(* Close file and validate data *)
SysFileClose(File:=hFile);
END_ACTION
ACTION DB_SetName:
(* Create current filename 'yyyyCRnn.DAT' *)
sFile:=CONCAT(FilesPath,WORD_TO_STRING(Sys.Time_Year));
sFile:=CONCAT(STR1:=sFile, STR2:='CR');
IF ID<10 THEN
sFile:=CONCAT(STR1:=sFile, STR2:='0');
END_IF
sFile:=CONCAT(STR1:=sFile, STR2:=BYTE_TO_STRING(ID));
sFile:=CONCAT(STR1:=sFile, STR2:='.DAT');
END_ACTION
ACTION Init:
DB_Load();
InitOK:=TRUE;
END_ACTION

(* POU Plant_Objects/obj_CTL, ST *)
FUNCTION_BLOCK obj_CTL
(* === PULSE VOLUME COUNTER ===
   v1.0[16/04/15] - Versioning
*)
VAR_INPUT
	(* Settings *)
	ID				: BYTE;	(* Index of instanced object *)
	Peso			: DWORD;
	(* Physical inputs *)
	CTL_ST			: BOOL;
END_VAR
VAR_IN_OUT
	COUNT			: DWORD;
END_VAR
VAR_OUTPUT
	(* Status *)
	Status_Log		: BYTE;
END_VAR
VAR
	Filter			: FLT_TAP := ( INITEV:=FALSE );
	Timer			: TON;
	TCount			: DWORD;
	i				: DWORD;
END_VAR
(* Execute timer *)
Timer(IN:=NOT Timer.Q, PT:=T#60m);

(* Execute filter on counter status *)
Filter(IN:=CTL_ST);

(* Count event *)
IF Filter.EVH THEN
	COUNT:=COUNT+Peso;
	TCount:=TCount+1;
	(* Check flow rate *)
	IF TCount>=Plant_MaxWaterLoss THEN
		i:=(TCount*TIME_TO_DWORD(Timer.PT))/TIME_TO_DWORD(Timer.ET);	(* Estimated mc per hour *)
		i:= i * Peso;

		(* NB The weight is multiplied by 10 -> Need to divide it by 10 server side *)
		LogEv(EL_AlarmStop,EO_CTL,ID,1,DWORD_TO_STRING(i));
		Status_Log:=2;

		TCount:=0;
		Timer(IN:=FALSE);
	END_IF
END_IF
(* Check timer *)
IF Timer.Q THEN
	TCount:=0;							(* One hour is elapsed *)
	IF TCount<Plant_MaxWaterLoss THEN
		Status_Log:=0;
	END_IF
END_IF
END_FUNCTION_BLOCK
ACTION AddLogData:
Logger.s1:=INSERT('&CTL=',BYTE_TO_STRING(ID),4);
IF ID<10 THEN Logger.s1:=INSERT(Logger.s1,'0',4); END_IF

Logger.s1:=CONCAT(Logger.s1,DWORD_TO_STRING(COUNT));			Logger.s1:=CONCAT(Logger.s1,';');

Logger.s1:=CONCAT(Logger.s1,WORD_TO_STRING(Status_Log));
ADDSTRING(ADR(Logger.TData), ADR(Logger.s1), Logger.TLen);
END_ACTION

(* POU Plant_Objects/obj_MODBUS, ST *)
FUNCTION_BLOCK obj_MODBUS
(* === MODBUS PROTOCOL INTERFACE ===
   v1.1[19/06/15] - Added new VARS allocation and searching
*)
VAR CONSTANT
	VARS_Max	: BYTE := 32;
END_VAR
VAR_INPUT
	(* Settings *)
	ID			: BYTE;
	COM			: BYTE;
	BAUDRATE	: COM_BAUDRATE;
	RS485		: BOOL := FALSE;

	N_STOPBits	:BYTE:=1;

	(* Interface *)
	MB_MASTER	: MODBUS_EXTENDED_MASTER;
	MB_Start	: BOOL;
	MB_Query	: typModbusExtendedQuery;
	MB_Resp		: typModbusResponse;
	MB_Lock		: BOOL;
	MB_timeOut	: TIME := t#500ms;

	(* Variables management *)
	VARS_En		: BOOL;
	VARS		: ARRAY [0..VARS_Max] OF typ_MODBUS_VAR;
	VARS_Check	: BOOL;
	VARS_Alarm	: BOOL;

	(* Variables allocation *)
	VAR_Pointer : POINTER TO ARRAY[0..99] OF WORD;
	VAR_Cfg		: POINTER TO typ_MODBUS_VAR;
END_VAR
VAR_OUTPUT
	(* Status *)
	Status_Log	: BYTE;
	Status_Vis	: DWORD;
END_VAR
VAR
	sta         : BYTE :=0;
	i			: BYTE;
	j			: BYTE;
	Alarm		: FLT_EVENT;
	
	VarTmr		: TON := (PT:=T#1s);
	VarSta		: BYTE; (* Status *)
	VarCnt		: BYTE; (* Scan counter *)
	VarRetry	: BYTE;
	VarAlarm	: BYTE; (* Last variable with errors *)
END_VAR
IF N_STOPBits=1 THEN MB_MASTER.csCOM_STOPBITS:=STOPBITS_1;END_IF
IF N_STOPBits=2 THEN MB_MASTER.csCOM_STOPBITS:=STOPBITS_2;END_IF


(** PARITY_NO **)



MB_MASTER(ENABLE:=TRUE,	ASCII_Mode:=FALSE, bCOM_PORT:=COM, cbCOM_BAUDRATE:=BAUDRATE, cpCOM_PARITY:=PARITY_EVEN,
		cbsCOM_BYTESIZE:=BS_8, cfCOM_FLOW_CONTROL:=SEL(RS485,NO_FLOW_CONTROL,HALFDUPLEX),
		tTIME_OUT:=MB_timeOut,	StartFunction:=MB_Start, ExtQuery:=MB_Query, Response:=MB_Resp);

(* Process variable management *)
IF VARS_En THEN VARS_Process(); END_IF

(* Check status *)
Alarm(IN:=(MB_MASTER.bInterfaceError<>0));
IF Alarm.EVH THEN
	LogEv(SEL(MB_MASTER.bInterfaceError<>3,EL_Wrn,EL_Alarm),EO_MODBUS,ID,1,BYTE_TO_STRING(MB_MASTER.bInterfaceError));
END_IF
IF Alarm.EVL THEN								(* Trigger a fall edge: MODBUS back working *)
	LogEv(EL_Log,EO_MODBUS,ID,2,'MODBUS_OK');
END_IF

(* Log/visu status *)
   IF Alarm.IN   THEN Status_Log:=2; Status_Vis:=COLOR_RED;
ELSIF Vars_Alarm THEN Status_Log:=1; Status_Vis:=COLOR_YELLOW;
  				 ELSE Status_Log:=0; Status_Vis:=COLOR_GREEN;
END_IF
END_FUNCTION_BLOCK
ACTION VAR_Search:
(* Search VAR with specific pointer if not found return first free VAR
	[Last VAR is not active... used as safe area...] 
*)
j:=VARS_Max;
FOR i := 0 TO VARS_Max-1 DO
	IF VARS[i].Variable=0 AND j>i THEN j:=i; END_IF
	IF VARS[i].Variable=VAR_Pointer THEN
		VAR_Cfg:=ADR(VARS[i]);
		RETURN;
	END_IF
END_FOR
VAR_Cfg:=ADR(VARS[j]);
END_ACTION
ACTION VARS_Process:
(* Update var timers *)
VarTmr(IN:=(NOT VarTmr.Q));
IF VarTmr.Q THEN
	FOR i := 0 TO VARS_Max DO
		IF VARS[i].Refresh_Cnt>0 THEN VARS[i].Refresh_Cnt:=VARS[i].Refresh_Cnt-1; END_IF
	END_FOR
	VARS_Check:=TRUE;
END_IF


(* Process status *)
CASE VarSta OF
	0: (* === Init *)
		VarCnt:=0;
		VarSta:=1;

	1: (* === Wait check signal *)
		IF VARS_Check THEN				(* Decremented "Refresh_Cnt" *)
			VARS_Check:=FALSE;
			VarCnt:=0;
			VarSta:=2;
		END_IF

	2: (* === Check loop *)
		IF NOT (MB_Lock OR MB_Start) THEN
			WHILE VarCnt<=(VARS_Max-1) AND VarSta=2 DO
				(* Check only active vars *)
				IF VARS[VarCnt].Variable<>0 THEN			(* "Variable" is a pointer to word, so if 0 no address *)
					(* Check var auto-refresh on timer checks *)
					IF VARS[VarCnt].Refresh_Time>0 AND VARS[VarCnt].Refresh_Cnt=0 THEN
						VARS[VarCnt].Refresh_Cnt:=VARS[VarCnt].Refresh_Time;
						VarSta:=3;
					END_IF
					(* Check refresh for change or request *)
					CASE VARS[VarCnt].FunCode OF
						5,6,15,16: (* Write functions *)
							IF VARS[VarCnt].Variable_Size=1 THEN
								IF VARS[VarCnt].Variable^<>VARS[VarCnt].Variable_Mirror THEN
									VARS[VarCnt].Variable_Mirror:=VARS[VarCnt].Variable^;
									VarSta:=3;
								END_IF
							ELSE
								IF VARS[VarCnt].Variable_Mirror<>0 THEN
									VARS[VarCnt].Variable_Mirror:=0;
									VarSta:=3;
								END_IF
							END_IF
						1,2,3,4: (* Read functions *)
							IF VARS[VarCnt].Variable_Mirror<>0 THEN
								VARS[VarCnt].Variable_Mirror:=0;
								VarSta:=3;
							END_IF
					END_CASE
				END_IF
				(* Process query *)
				IF VarSta=3 THEN
					MB_Lock:=TRUE;
					MB_Query.SlaveAddress:=VARS[VarCnt].SlaveAddress;
					MB_Query.FunctionCode:=VARS[VarCnt].FunCode;
					CASE VARS[VarCnt].FunCode OF
						16#5,16#6,16#F,16#10:
							MB_Query.Read_Quantity:=0;
							MB_Query.Read_StartAddress:=0;
							MB_Query.Write_StartAddress:=VARS[VarCnt].FunAddress;
							MB_Query.Write_Quantity:=VARS[VarCnt].Variable_Size;
							IF VARS[VarCnt].Variable_Size=200 THEN
								COPY_32SWAP16(VARS[VarCnt].Variable, ADR(MB_Query.Write_Data[0]));
							ELSIF VARS[VarCnt].Variable_Size>1 THEN
								MEMCPY(VARS[VarCnt].Variable, ADR(MB_Query.Write_Data[0]), 2*VARS[VarCnt].Variable_Size);
							ELSE
								MB_Query.Write_Data[0]:=VARS[VarCnt].Variable^;
							END_IF
						16#1,16#2,16#3,16#4:
							MB_Query.Read_StartAddress:=VARS[VarCnt].FunAddress;
							IF VARS[VarCnt].Variable_Size=200 THEN MB_Query.Read_Quantity:=2; ELSE
							  MB_Query.Read_Quantity:=VARS[VarCnt].Variable_Size;
							END_IF
							MB_Query.Write_StartAddress:=0;
							MB_Query.Write_Quantity:=0;
					END_CASE
					VarRetry:=0;
					MB_Start:=TRUE;
				ELSE
					VarCnt:=VarCnt+1;
				END_IF
			END_WHILE
			(* Check loop completed -> no actions *)
			IF VarSta=2 THEN VarSta:=1; END_IF
		END_IF

	3: (* === Wait & process MB response *)
		IF NOT MB_Start THEN
			IF MB_MASTER.MB_Error=0 THEN
				CASE VARS[VarCnt].FunCode OF
					1,2,3,4:
						IF VARS[VarCnt].Variable_Size=200 THEN
							COPY_32SWAP16(ADR(MB_Resp.Data), VARS[VarCnt].Variable);
						ELSIF VARS[VarCnt].Variable_Size>1 THEN
							MEMCPY(ADR(MB_Resp.Data), VARS[VarCnt].Variable, 2*VARS[VarCnt].Variable_Size);
						ELSE
							VARS[VarCnt].Variable^:=MB_Resp.Data[0];
						END_IF
				END_CASE
				MB_Lock:=FALSE;
				(* Signal error recovery *)
				IF VARS_Alarm=TRUE AND VarCnt=VarAlarm THEN
					LogEv(EL_Wrn,EO_MODBUS,ID,5,'');
					VARS_Alarm:=FALSE;
				END_IF
				(* Next var *)
				VarCnt:=VarCnt+1;
				VarSta:=2;
			ELSE
				IF VarRetry<3 THEN
					VarRetry:=VarRetry+1;
					MB_Start:=TRUE;
				ELSE
					MB_Lock:=FALSE;
					(* Signal error *)
					IF VARS_Alarm=FALSE THEN
						LogEv(EL_Wrn,EO_MODBUS,ID,3,INT_TO_STRING(MB_MASTER.MB_Error));
						VARS_Alarm:=TRUE;
						VarAlarm:=VarCnt-1;
					END_IF
					(* Next var *)
					VarCnt:=VarCnt+1;
					VarSta:=2;
				END_IF
			END_IF
		END_IF

ELSE
	VarSta:=0;
END_CASE
END_ACTION

(* POU Plant_Objects/obj_MODBUS_THAITY_ELECTA, ST *)
FUNCTION_BLOCK obj_MODBUS_THAITY_ELECTA
VAR CONSTANT
	TimeOutModBus: TON;

END_VAR
VAR_INPUT
	ID			:	BYTE;
	Address		:	BYTE;


	SetPointManuale: INT; 			(* SetPoint forazato in manuale escludendo la curva di carico *)
	AbilitaSetPointManuale : BOOL ; (* Abilita il funzionamento col set point Manaule Escludendo la curva cliamtica *)


	(* Modbus *)
	Refresh_Now	:	BOOL;			(* Richiesta di lettura stato macchina Immediata  *)
	retryErrMax	:	BYTE := 2;

	Temperatura: INT;


	STOP_REQ: BOOL;
	RUN_REQ: BOOL;
	(* Timings *)
	OnDelay		:	TIME;
	OffDelay	:	TIME;

	OnOff		: 	BOOL;

	IndirizzoDaScrivere: WORD;
	DatoDaScrivere: INT;
	ScriviDato: BOOL;
	ScriviCoil: BOOL;


	ImpMB_2SetPoint: INT;
	ImpMB_ResetFrigo: BOOL;
	ImpMB_LocRem: BOOL;
	fWriteAttivazioneComandi:BOOL;




END_VAR
VAR_IN_OUT
	ModBus		:obj_MODBUS;
	CLIM		:typ_Clima;

END_VAR
VAR_OUTPUT
	Run			:	BOOL;

	Status_Log	:	WORD;
	Status_Vis	:	DWORD;
END_VAR
VAR
	(* da diego per gestione stato stringa > 255*)
	temp :STRING(255);
	tempRaw		: ARRAY [0..MAX_SEND_TCP_CLIENT] OF BYTE;
	tempRawLen :DINT;
	longString :STRING(250);

	(* Timer manage switch on/off delay *)
	Delay		: 	TONOF;

	AllarmePDC_MB		:ARRAY [1..11] OF	FLT_EVENT;
	AllarmePDC: BOOL;

	AllarmeRemotoFLT:	FLT_EVENT;
	AllarmeRemoto: BOOL;

	state		:	INT;
	retry		:	BYTE;
	retryErr	:	BYTE;
	ReadTmr		:	TON := (PT:=T#5s);
	fModbusAlr:BOOL;

(*	retry_write	:	BYTE;
	fWriteStatus:	BOOL;
	fWriteMode	:	BOOL;
	fWriteReset	:	BOOL; *)

	SetPointCC: DINT;
	x: INT;
	ImpMB_SetPoint: INT;
	Ctrl_Run: BOOL;


	VerificaFuctionCode: INT;
	VerificaNodoLetto: INT;
	ErroreComuModBus: BOOL;
	IndiceErrore: BYTE;

	MB_BitStato: ARRAY [0..200] OF BOOL;
	MB_RegistriLetti: ARRAY [0..450] OF INT;
	MB_Moreno: ARRAY [0..450] OF INT;

	AddressRead: BYTE;
	index: BYTE;
	indexErr: BYTE;


	indirizzoDaleggere: INT;
END_VAR
(* Aggiornamento in tempo reale dei TON e TOFF funzionamento Pompa *)

Delay.PT_OF := OffDelay;
Delay.PT_ON := OnDelay + WORD_TO_TIME(1000*ID);

(* Check climatic setup *)
IF NOT CLIM.InitOK THEN Clima_Default(); END_IF;
(* Calculate Setpoint *)

	IF Temperatura>=CLIM.Points[0].X  THEN SetPointCC:=CLIM.Points[0].Y; END_IF;
	IF Temperatura>=CLIM.Points[1].X AND Temperatura<CLIM.Points[0].X THEN SetPointCC:=CLIM.Points[0].Y; END_IF;
	IF Temperatura>=CLIM.Points[2].X AND Temperatura<CLIM.Points[1].X THEN SetPointCC:=CLIM.Points[1].Y; END_IF;
	IF Temperatura>=CLIM.Points[3].X AND Temperatura<CLIM.Points[2].X THEN SetPointCC:=CLIM.Points[2].Y; END_IF;
	IF Temperatura>=CLIM.Points[4].X AND Temperatura<CLIM.Points[3].X THEN SetPointCC:=CLIM.Points[3].Y; END_IF;
	IF Temperatura<CLIM.Points[4].X THEN SetPointCC:=CLIM.Points[4].Y; END_IF;


	IF Temperatura<CLIM.Points[4].X THEN SetPointCC:=CLIM.Points[4].Y; END_IF;


(* Scelta del set point della cladaia o vien preso dalla curva cliamtica o da un riferimento esterno *)
IF AbilitaSetPointManuale THEN
	ImpMB_SetPoint:=(SetPointManuale);
ELSE
	ImpMB_SetPoint:=DINT_TO_INT(SetPointCC);
END_IF


(* Controllo Bit di funzionamento ON e OFF  *)
Ctrl_Run := OnOff;
Delay(IN:=Ctrl_Run);



IF STOP_REQ THEN Run := 1;
	ELSIF RUN_REQ THEN Run := 0;
ELSE
	Run :=Delay.OUT;
END_IF



(* Call ModBus state machine *)
Stm();

(* Check alarm	*)
CheckAlarm();
END_FUNCTION_BLOCK
ACTION AddLogData:
Logger.s1:=INSERT('&PDC=',BYTE_TO_STRING(ID),4);
IF ID<10 THEN Logger.s1:=INSERT(Logger.s1,'0',4); END_IF



Logger.s1:=CONCAT(Logger.s1,INT_TO_STRING(MB_RegistriLetti[20]));
Logger.s1:=CONCAT(Logger.s1,';');

Logger.s1:=CONCAT(Logger.s1,SEL(WORD_TO_BOOL(MB_RegistriLetti[34]),'0','100'));
Logger.s1:=CONCAT(Logger.s1,';');

Logger.s1:=CONCAT(Logger.s1,WORD_TO_STRING(Status_Log));
ADDSTRING(ADR(Logger.TData), ADR(Logger.s1), Logger.TLen);









(*
FOR tempRawLen:=0 TO MAX_SEND_TCP_CLIENT DO
                tempRaw[tempRawLen]:=0;
END_FOR

tempRawLen:=0;


temp:=Logger.s1;
ADDSTRING(ADR(tempRaw), ADR(temp), tempRawLen);

FOR x:= 1 TO 46 DO

	temp:=CONCAT(INT_TO_STRING(MB_RegistriLetti[x]),';');
	ADDSTRING(ADR(tempRaw), ADR(temp), tempRawLen);

END_FOR

temp:=CONCAT(temp,WORD_TO_STRING(Status_Log));

ADDSTRING(ADR(tempRaw), ADR(temp), tempRawLen);
ADDSTRING(ADR(Logger.TData), ADR(tempRaw), Logger.TLen); *)
END_ACTION
ACTION CheckAlarm:
(**** GEstione Log ad Evento *****)


FOR x:=1 TO 10 DO

	AllarmePDC_MB[x](IN:=WORD_TO_BOOL(MB_RegistriLetti[x+22]) );

	IF AllarmePDC_MB[x].EVH THEN
		LogEv(EL_Alarm,EO_PDC,ID,x,CONCAT ('Allarme Attivo n. ', INT_TO_STRING(x)));
	END_IF

	IF AllarmePDC_MB[x].EVL THEN
		LogEv(EL_Log,EO_PDC,ID,x,CONCAT ('Allarme Rientrato n. ', INT_TO_STRING(x)));
	END_IF

END_FOR


AllarmePDC:=FALSE;
FOR x:=1 TO 10 DO
	IF AllarmePDC_MB[x].IN THEN
		AllarmePDC:=TRUE;
	END_IF
END_FOR


	AllarmeRemotoFLT(IN:=WORD_TO_BOOL(MB_RegistriLetti[6]) );

	IF AllarmeRemotoFLT.EVH THEN
		LogEv(EL_Alarm,EO_PDC,ID,11,'Controllo_Remoto_OK');
		AllarmeRemoto:=FALSE;
	END_IF

	IF AllarmeRemotoFLT.EVL THEN
		LogEv(EL_Alarm,EO_PDC,ID,12,'Controllo_Locale_Fault');
		AllarmeRemoto:=TRUE;
	END_IF





(* Seganalzione stato Frigorifero  *)
IF ErroreComuModBus OR AllarmePDC OR AllarmeRemoto THEN
		Status_Log:=2;
		Status_Vis:=16#2020F0;
    ELSE
		Status_Log:=0;
		Status_Vis:=16#006000;
END_IF
END_ACTION
ACTION Clima_Default:
IF CLIM.Points[0].X=0 THEN
	CLIM.Points[0].X:=-300; CLIM.Points[0].Y:=770;
	CLIM.Points[1].X:=-70 ; CLIM.Points[1].Y:=770;
	CLIM.Points[2].X:= 80; 	CLIM.Points[2].Y:=690;
	CLIM.Points[3].X:= 200; CLIM.Points[3].Y:=300;
	CLIM.Points[4].X:= 500; CLIM.Points[4].Y:=200;
END_IF
CLIM.InitOK:=TRUE;
LogEv(EL_Wrn,EO_PDC,ID,0,'Climatic_default');
END_ACTION
ACTION Stm:
CASE state OF
	0:	(* Refresh time manager *)
		ReadTmr(IN:=NOT ReadTmr.Q);
		(*A tempo interrogo il nodo sempre che non ci sia qualcuno che lo sta interrogando in quel momento *)

		IF (ReadTmr.Q AND NodoDaInterrogarePDC=Address )OR Refresh_Now AND NOT InibiscoModbusPDC THEN
			state := 10;
			ReadTmr.PT := T#5s;  (* moreno *)
			Refresh_Now := FALSE;
			InibiscoModbusPDC := TRUE;
		END_IF

	(**** Leggo le Analogiche a Disposzione  ****)

	10:	(* richiedo lettura Holding Registere Chiller  *)

		Modbus.MB_Query.SlaveAddress := Address;
		Modbus.MB_Query.FunctionCode := 3;
		ModBus.MB_Query.Read_StartAddress := 8975 ;			(* richiedo lettura altri Parametri *)
		ModBus.MB_Query.Read_Quantity := 10;
		ModBus.MB_Start := TRUE;
		state := 20;

	20:	(* Risposta all'interrogazione *)
		IF NOT ModBus.MB_Start   THEN
			VerificaFuctionCode:=ModBus.MB_Resp.FunctionCode;
			VerificaNodoLetto:=ModBus.MB_Resp.SlaveAddress;

			IF ModBus.MB_MASTER.MB_Error<>0 THEN
				state := 300;
			ELSE
				MB_RegistriLetti[1] := ModBus.MB_Resp.Data[0];   	(* Vedi tabella *)
				MB_RegistriLetti[2] := ModBus.MB_Resp.Data[1];		(* Vedi tabella *)

				ModBus.MB_Query.Read_StartAddress := 8961; 	(* richiedo lettura altri Parametri *)
				ModBus.MB_Query.Read_Quantity := 18;
				ModBus.MB_Start := TRUE;

				state := 30;
			END_IF
		END_IF

	30: (* Rispota Altri paramenti *)
		IF NOT ModBus.MB_Start  THEN

			IF ModBus.MB_MASTER.MB_Error<>0 THEN
				state := 300;
			ELSE
				MB_RegistriLetti[3] := ModBus.MB_Resp.Data[0];   	(* Vedi tabella *)
				MB_RegistriLetti[4] := ModBus.MB_Resp.Data[1];		(* Vedi tabella *)
				MB_RegistriLetti[5] := ModBus.MB_Resp.Data[3];		(* Vedi tabella *)
				MB_RegistriLetti[6] := ModBus.MB_Resp.Data[4];		(* Vedi tabella *)
				MB_RegistriLetti[7] := ModBus.MB_Resp.Data[5];		(* Vedi tabella *)
				MB_RegistriLetti[8] := ModBus.MB_Resp.Data[7];		(* Vedi tabella *)
				MB_RegistriLetti[9] := ModBus.MB_Resp.Data[9];		(* Vedi tabella *)
				MB_RegistriLetti[10] := ModBus.MB_Resp.Data[10];		(* Vedi tabella *)
				MB_RegistriLetti[11] := ModBus.MB_Resp.Data[11];		(* Vedi tabella *)
				MB_RegistriLetti[12] := ModBus.MB_Resp.Data[12];		(* Vedi tabella *)
				MB_RegistriLetti[13] := ModBus.MB_Resp.Data[16];		(* Vedi tabella *)

				ModBus.MB_Query.Read_StartAddress := 8983; (* richiedo lettura altri Parametri *)
				ModBus.MB_Query.Read_Quantity := 20;
				ModBus.MB_Start := TRUE;

				state := 40;
			END_IF
		END_IF

	40: (* Rispota Altri paramenti *)
		IF NOT ModBus.MB_Start  THEN

			IF ModBus.MB_MASTER.MB_Error<>0 THEN
				state := 300;
			ELSE
				MB_RegistriLetti[14] := ModBus.MB_Resp.Data[0];   	(* Vedi tabella *)
				MB_RegistriLetti[15] := ModBus.MB_Resp.Data[2];		(* Vedi tabella *)
				MB_RegistriLetti[16] := ModBus.MB_Resp.Data[6];		(* Vedi tabella *)
				MB_RegistriLetti[17] := ModBus.MB_Resp.Data[7];		(* Vedi tabella *)
				MB_RegistriLetti[18] := ModBus.MB_Resp.Data[8];		(* Vedi tabella *)
				MB_RegistriLetti[19] := ModBus.MB_Resp.Data[9];		(* Vedi tabella *)
				MB_RegistriLetti[20] := ModBus.MB_Resp.Data[10];		(* Vedi tabella *)
				MB_RegistriLetti[21] := ModBus.MB_Resp.Data[13];		(* Vedi tabella *)
				MB_RegistriLetti[22] := ModBus.MB_Resp.Data[17];		(* Vedi tabella *)

				ModBus.MB_Query.Read_StartAddress := 9003; (* richiedo lettura altri Parametri *)
				ModBus.MB_Query.Read_Quantity := 12;
				ModBus.MB_Start := TRUE;

				state := 45;
			END_IF
		END_IF

	45: (* Rispota Altri paramenti *)
		IF NOT ModBus.MB_Start  THEN

			IF ModBus.MB_MASTER.MB_Error<>0 THEN
				state := 300;
			ELSE
				MB_RegistriLetti[23] := ModBus.MB_Resp.Data[0];   	(* Vedi tabella *)
				MB_RegistriLetti[24] := ModBus.MB_Resp.Data[1];		(* Vedi tabella *)
				MB_RegistriLetti[25] := ModBus.MB_Resp.Data[2];		(* Vedi tabella *)
				MB_RegistriLetti[26] := ModBus.MB_Resp.Data[3];		(* Vedi tabella *)
				MB_RegistriLetti[27] := ModBus.MB_Resp.Data[4];		(* Vedi tabella *)
				MB_RegistriLetti[28] := ModBus.MB_Resp.Data[5];		(* Vedi tabella *)
				MB_RegistriLetti[29] := ModBus.MB_Resp.Data[6];		(* Vedi tabella *)
				MB_RegistriLetti[30] := ModBus.MB_Resp.Data[7];		(* Vedi tabella *)
				MB_RegistriLetti[31] := ModBus.MB_Resp.Data[9];		(* Vedi tabella *)
				MB_RegistriLetti[32] := ModBus.MB_Resp.Data[10];		(* Vedi tabella *)

				ModBus.MB_Query.Read_StartAddress := 16383; (* richiedo lettura altri Parametri *)
				ModBus.MB_Query.Read_Quantity := 20;
				ModBus.MB_Start := TRUE;

				state := 50;
			END_IF
		END_IF
	50: (* Rispota Altri paramenti *)
		IF NOT ModBus.MB_Start  THEN

			IF ModBus.MB_MASTER.MB_Error<>0 THEN
				state := 300;
			ELSE
				MB_RegistriLetti[33] := ModBus.MB_Resp.Data[0];   	(* Vedi tabella *)
				MB_RegistriLetti[34] := ModBus.MB_Resp.Data[1];		(* Vedi tabella *)
				MB_RegistriLetti[35] := ModBus.MB_Resp.Data[2];		(* Vedi tabella *)
				MB_RegistriLetti[36] := ModBus.MB_Resp.Data[3];		(* Vedi tabella *)
				MB_RegistriLetti[37] := ModBus.MB_Resp.Data[4];		(* Vedi tabella *)
				MB_RegistriLetti[38] := ModBus.MB_Resp.Data[5];		(* Vedi tabella *)
				MB_RegistriLetti[39] := ModBus.MB_Resp.Data[6];		(* Vedi tabella *)
				MB_RegistriLetti[40] := ModBus.MB_Resp.Data[8];		(* Vedi tabella *)
				MB_RegistriLetti[41] := ModBus.MB_Resp.Data[9];		(* Vedi tabella *)
				MB_RegistriLetti[42] := ModBus.MB_Resp.Data[11];		(* Vedi tabella *)
				MB_RegistriLetti[43] := ModBus.MB_Resp.Data[12];		(* Vedi tabella *)
				MB_RegistriLetti[44] := ModBus.MB_Resp.Data[13];		(* Vedi tabella *)
				MB_RegistriLetti[45] := ModBus.MB_Resp.Data[14];		(* Vedi tabella *)
				MB_RegistriLetti[46] := ModBus.MB_Resp.Data[15];		(* Vedi tabella *)

				ModBus.MB_Query.Read_StartAddress := 16399; (* richiedo lettura altri Parametri *)
				ModBus.MB_Query.Read_Quantity := 20;
				ModBus.MB_Start := TRUE;

				state := 55;
			END_IF
		END_IF

	55: (* Rispota Altri paramenti *)
		IF NOT ModBus.MB_Start  THEN

			IF ModBus.MB_MASTER.MB_Error<>0 THEN
				state := 300;
			ELSE
				MB_RegistriLetti[47] := ModBus.MB_Resp.Data[0];   	(* Vedi tabella *)
				MB_RegistriLetti[48] := ModBus.MB_Resp.Data[1];		(* Vedi tabella *)
				MB_RegistriLetti[49] := ModBus.MB_Resp.Data[2];		(* Vedi tabella *)
				MB_RegistriLetti[50] := ModBus.MB_Resp.Data[3];		(* Vedi tabella *)
				MB_RegistriLetti[51] := ModBus.MB_Resp.Data[4];		(* Vedi tabella *)
				MB_RegistriLetti[52] := ModBus.MB_Resp.Data[5];		(* Vedi tabella *)
				MB_RegistriLetti[53] := ModBus.MB_Resp.Data[6];		(* Vedi tabella *)
				MB_RegistriLetti[54] := ModBus.MB_Resp.Data[7];		(* Vedi tabella *)
				MB_RegistriLetti[55] := ModBus.MB_Resp.Data[8];		(* Vedi tabella *)
				MB_RegistriLetti[56] := ModBus.MB_Resp.Data[9];		(* Vedi tabella *)
				MB_RegistriLetti[57] := ModBus.MB_Resp.Data[10];		(* Vedi tabella *)
				MB_RegistriLetti[58] := ModBus.MB_Resp.Data[11];		(* Vedi tabella *)
				MB_RegistriLetti[59] := ModBus.MB_Resp.Data[12];		(* Vedi tabella *)
				MB_RegistriLetti[60] := ModBus.MB_Resp.Data[13];		(* Vedi tabella *)
				MB_RegistriLetti[61] := ModBus.MB_Resp.Data[14];		(* Vedi tabella *)
				MB_RegistriLetti[62] := ModBus.MB_Resp.Data[15];		(* Vedi tabella *)
				MB_RegistriLetti[63] := ModBus.MB_Resp.Data[16];		(* Vedi tabella *)
				MB_RegistriLetti[64] := ModBus.MB_Resp.Data[17];		(* Vedi tabella *)
				MB_RegistriLetti[65] := ModBus.MB_Resp.Data[18];		(* Vedi tabella *)
				MB_RegistriLetti[66] := ModBus.MB_Resp.Data[19];		(* Vedi tabella *)

				ModBus.MB_Query.Read_StartAddress := 16419; (* richiedo lettura altri Parametri *)
				ModBus.MB_Query.Read_Quantity := 20;
				ModBus.MB_Start := TRUE;

				state := 60;
			END_IF
		END_IF

	60: (* Rispota Altri paramenti *)
		IF NOT ModBus.MB_Start  THEN

			IF ModBus.MB_MASTER.MB_Error<>0 THEN
				state := 300;
			ELSE
				MB_RegistriLetti[67] := ModBus.MB_Resp.Data[0];   	(* Vedi tabella *)
				MB_RegistriLetti[68] := ModBus.MB_Resp.Data[1];		(* Vedi tabella *)
				MB_RegistriLetti[69] := ModBus.MB_Resp.Data[2];		(* Vedi tabella *)
				MB_RegistriLetti[70] := ModBus.MB_Resp.Data[3];		(* Vedi tabella *)
				MB_RegistriLetti[71] := ModBus.MB_Resp.Data[4];		(* Vedi tabella *)
				MB_RegistriLetti[72] := ModBus.MB_Resp.Data[5];		(* Vedi tabella *)
				MB_RegistriLetti[73] := ModBus.MB_Resp.Data[6];		(* Vedi tabella *)
				MB_RegistriLetti[74] := ModBus.MB_Resp.Data[7];		(* Vedi tabella *)
				MB_RegistriLetti[75] := ModBus.MB_Resp.Data[8];		(* Vedi tabella *)
				MB_RegistriLetti[76] := ModBus.MB_Resp.Data[9];		(* Vedi tabella *)
				MB_RegistriLetti[77] := ModBus.MB_Resp.Data[10];		(* Vedi tabella *)
				MB_RegistriLetti[78] := ModBus.MB_Resp.Data[11];		(* Vedi tabella *)
				MB_RegistriLetti[79] := ModBus.MB_Resp.Data[12];		(* Vedi tabella *)
				MB_RegistriLetti[80] := ModBus.MB_Resp.Data[13];		(* Vedi tabella *)
				MB_RegistriLetti[81] := ModBus.MB_Resp.Data[14];		(* Vedi tabella *)
				MB_RegistriLetti[82] := ModBus.MB_Resp.Data[15];		(* Vedi tabella *)
				MB_RegistriLetti[83] := ModBus.MB_Resp.Data[16];		(* Vedi tabella *)

				ModBus.MB_Query.Read_StartAddress := 16442; (* richiedo lettura altri Parametri *)
				ModBus.MB_Query.Read_Quantity := 10;
				ModBus.MB_Start := TRUE;

				state := 65;
			END_IF
		END_IF

	65: (* Rispota Altri paramenti *)
		IF NOT ModBus.MB_Start  THEN

			IF ModBus.MB_MASTER.MB_Error<>0 THEN
				state := 300;
			ELSE
				MB_RegistriLetti[84] := ModBus.MB_Resp.Data[0];   	(* Vedi tabella *)
				MB_RegistriLetti[85] := ModBus.MB_Resp.Data[1];		(* Vedi tabella *)
				MB_RegistriLetti[86] := ModBus.MB_Resp.Data[2];		(* Vedi tabella *)
				MB_RegistriLetti[87] := ModBus.MB_Resp.Data[3];		(* Vedi tabella *)
				MB_RegistriLetti[88] := ModBus.MB_Resp.Data[4];		(* Vedi tabella *)

				ModBus.MB_Query.Read_StartAddress := 16451; (* richiedo lettura altri Parametri *)
				ModBus.MB_Query.Read_Quantity := 20;
				ModBus.MB_Start := TRUE;

				state := 70;
			END_IF
		END_IF

	70: (* Rispota Altri paramenti *)
		IF NOT ModBus.MB_Start  THEN

			IF ModBus.MB_MASTER.MB_Error<>0 THEN
				state := 300;
			ELSE
				MB_RegistriLetti[89] := ModBus.MB_Resp.Data[0];   	(* Vedi tabella *)
				MB_RegistriLetti[90] := ModBus.MB_Resp.Data[1];		(* Vedi tabella *)
				MB_RegistriLetti[91] := ModBus.MB_Resp.Data[2];		(* Vedi tabella *)
				MB_RegistriLetti[92] := ModBus.MB_Resp.Data[3];		(* Vedi tabella *)
				MB_RegistriLetti[93] := ModBus.MB_Resp.Data[4];		(* Vedi tabella *)
				MB_RegistriLetti[94] := ModBus.MB_Resp.Data[5];		(* Vedi tabella *)
				MB_RegistriLetti[95] := ModBus.MB_Resp.Data[6];		(* Vedi tabella *)
				MB_RegistriLetti[96] := ModBus.MB_Resp.Data[7];		(* Vedi tabella *)
				MB_RegistriLetti[97] := ModBus.MB_Resp.Data[8];		(* Vedi tabella *)
				MB_RegistriLetti[98] := ModBus.MB_Resp.Data[9];		(* Vedi tabella *)
				MB_RegistriLetti[99] := ModBus.MB_Resp.Data[10];		(* Vedi tabella *)
				MB_RegistriLetti[100] := ModBus.MB_Resp.Data[11];		(* Vedi tabella *)
				MB_RegistriLetti[101] := ModBus.MB_Resp.Data[12];		(* Vedi tabella *)
				MB_RegistriLetti[102] := ModBus.MB_Resp.Data[13];		(* Vedi tabella *)
				MB_RegistriLetti[103] := ModBus.MB_Resp.Data[14];		(* Vedi tabella *)
				MB_RegistriLetti[104] := ModBus.MB_Resp.Data[15];		(* Vedi tabella *)
				MB_RegistriLetti[105] := ModBus.MB_Resp.Data[16];		(* Vedi tabella *)

				ModBus.MB_Query.Read_StartAddress := 16487; (* richiedo lettura altri Parametri *)
				ModBus.MB_Query.Read_Quantity := 2;
				ModBus.MB_Start := TRUE;

				state := 75;
			END_IF
		END_IF


	75: (* Rispota Altri paramenti *)
		IF NOT ModBus.MB_Start  THEN

			IF ModBus.MB_MASTER.MB_Error<>0 THEN
				state := 300;
			ELSE
				MB_RegistriLetti[106] := ModBus.MB_Resp.Data[0];   	(* Vedi tabella *)

				state := 200;
			END_IF
		END_IF



	100: (* Rispota Altri paramenti *)
		IF NOT ModBus.MB_Start  THEN

			IF ModBus.MB_MASTER.MB_Error<>0 THEN
				state := 300;
			ELSE
				ModBus.MB_Query.Read_StartAddress := indirizzoDaleggere; (* richiedo lettura altri Parametri *)
				ModBus.MB_Query.Read_Quantity := 4;
				ModBus.MB_Start := TRUE;

				state := 105;
			END_IF
		END_IF


	105: (* Rispota Altri paramenti *)
		IF NOT ModBus.MB_Start  THEN

			IF ModBus.MB_MASTER.MB_Error<>0 THEN
				state := 300;
			ELSE
				MB_Moreno[1] := ModBus.MB_Resp.Data[0];   	(* Vedi tabella *)
				MB_Moreno[2] := ModBus.MB_Resp.Data[1];		(* Vedi tabella *)
				MB_Moreno[3] := ModBus.MB_Resp.Data[2];		(* Vedi tabella *)
				MB_Moreno[4] := ModBus.MB_Resp.Data[3];		(* Vedi tabella *)

				state := 200;
			END_IF
		END_IF



	200:    (* Scrittura Abilitazione  *)
		IF NOT ModBus.MB_Start THEN
			IF ModBus.MB_MASTER.MB_Error<>0 THEN (*OR ModBus.MB_MASTER.MB_Error<>0 THEN*)
				state := 300;
			ELSE
					Modbus.MB_Query.FunctionCode := 6;
					Modbus.MB_Query.SlaveAddress := Address;
					ModBus.MB_Query.Write_StartAddress := 16384;
					ModBus.MB_Query.Write_Quantity :=1;
					ModBus.MB_Query.Write_Data[0] := BOOL_TO_WORD(Run);
					ModBus.MB_Start := TRUE;
					state := 210;
				END_IF
		END_IF

	210:    (* Scrittura Set Point  *)
		IF NOT ModBus.MB_Start THEN
			IF ModBus.MB_MASTER.MB_Error<>0 THEN (*OR ModBus.MB_MASTER.MB_Error<>0 THEN*)
				state := 300;
			ELSE
				IF Run <> INT_TO_BOOL (MB_RegistriLetti[34]) THEN
					Modbus.MB_Query.FunctionCode := 6;
					Modbus.MB_Query.SlaveAddress := Address;
					ModBus.MB_Query.Write_StartAddress := 16423;
					ModBus.MB_Query.Write_Quantity :=1;
					ModBus.MB_Query.Write_Data[0] := ImpMB_SetPoint+50;
					ModBus.MB_Start := TRUE;
					state := 215;
				ELSE
					state := 215;
				END_IF
			END_IF
		END_IF
	215:    (* Scrittura Set Point  *)
		IF NOT ModBus.MB_Start THEN
			IF ModBus.MB_MASTER.MB_Error<>0 THEN (*OR ModBus.MB_MASTER.MB_Error<>0 THEN*)
				state := 300;
			ELSE
				IF Run THEN
					Modbus.MB_Query.FunctionCode := 6;
					Modbus.MB_Query.SlaveAddress := Address;
					ModBus.MB_Query.Write_StartAddress := 16424;
					ModBus.MB_Query.Write_Quantity :=1;
					ModBus.MB_Query.Write_Data[0] := ImpMB_SetPoint+50;
					ModBus.MB_Start := TRUE;
					state := 290;
				ELSE
					state := 290;
				END_IF
			END_IF
		END_IF


		290:    (* Scrittura BOOL - COIL o WORD *)
		IF NOT ModBus.MB_Start THEN
			IF ModBus.MB_MASTER.MB_Error<>0 THEN (*OR ModBus.MB_MASTER.MB_Error<>0 THEN*)
				state := 300;
			ELSE
				IF ScriviDato THEN
				(*	IF ScriviCoil THEN
						Modbus.MB_Query.FunctionCode := 5;
					ELSE
						Modbus.MB_Query.FunctionCode := 6;
					END_IF *)
					Modbus.MB_Query.FunctionCode := 6;
					Modbus.MB_Query.SlaveAddress := Address;
					ModBus.MB_Query.Write_StartAddress := IndirizzoDaScrivere - 1;
					ModBus.MB_Query.Write_Quantity :=1;
					ModBus.MB_Query.Write_Data[0] := DatoDaScrivere;
					ModBus.MB_Start := TRUE;

				MB_Moreno[10] :=  MB_Moreno[10]+1;   	(* Vedi tabella *)

				(*		IF ScriviCoil THEN
							IF 	MB_BitStato[IndirizzoDaScrivere]=WORD_TO_BOOL(DatoDaScrivere) THEN
								ScriviDato:=FALSE;
							END_IF
						ELSE
							IF 	MB_RegistriLetti[IndirizzoDaScrivere]=DatoDaScrivere THEN
								ScriviDato:=FALSE;
							END_IF
						END_IF *)
					state := 295;
				ELSE
					state := 295;
				END_IF
			END_IF
		END_IF




		295:
		IF NOT ModBus.MB_Start THEN
			IF ModBus.MB_MASTER.MB_Error<>0 THEN (*OR ModBus.MB_MASTER.MB_Error<>0 THEN*)
				state := 300;
			ELSE
				IF fModbusAlr THEN fModbusAlr := FALSE; END_IF
				NodoDaInterrogarePDC:=Address+1;
				InibiscoModbusPDC:=FALSE;
				retryErr := 0;
				retry := 0;
				state := 0;
					IF fModbusAlr=FALSE AND ErroreComuModBus=TRUE THEN
						LogEv(EL_Log,EO_PDC,ID,62,'ComunicazioneModBus_OK');
						ErroreComuModBus := FALSE;
				(*	WarningCtr := SEL(WarningCtr=0, WarningCtr-1, 0); *)
					END_IF


			END_IF
		END_IF



	(**** CHECK MODBUS ERROR ****)
	300: 	(* Release MODBUS *)
			InibiscoModbusPDC:=FALSE;
			(* Retries *)
			retry:=retry+1;
			IF retry>3 THEN
				retry:=0;

				(* Verify if slave is dead *)
				IF retryErr < retryErrMaX THEN
					retryErr := retryErr + 1;
				ELSE
					fModbusAlr := TRUE;
					(* Verify ModBus error	*)

					IF fModbusAlr AND ErroreComuModBus=FALSE THEN
						LogEv(EL_Alarm,EO_PDC,ID,61,CONCAT('ErroreModbus_',INT_TO_STRING(ModBus.MB_MASTER.MB_Error)));
						ErroreComuModBus := TRUE;
					END_IF
				END_IF

				END_IF
			Refresh_Now := FALSE;
			NodoDaInterrogarePDC:=Address+1;
			state:=0;
END_CASE




(* Controllo Time Out Ciclo ModBus *)

TimeOutModBus(In:=state<>0,PT:=t#30s);
IF TimeOutModBus.Q THEN
	State:=0;
	Refresh_Now:=TRUE;  (* Rilancio la lettura del nodo *)
	IF MODBUS.MB_Lock=TRUE THEN MODBUS.MB_Lock:=FALSE;END_IF
	IF InibiscoModbusPDC=TRUE THEN InibiscoModbusPDC:=FALSE;END_IF
END_IF
END_ACTION

(* POU Plant_Objects/obj_TPV, ST *)
FUNCTION_BLOCK obj_TPV
(* === TEMPERATURE PROBE  ===
   v1.0[16/04/15] - Versioning
*)
VAR CONSTANT
	NormalEv		: BYTE := 0;
	ErrorEv			: BYTE := 1;
	WarningEv		: BYTE := 2;
END_VAR
VAR_INPUT
	(* Settings *)
	ID				: BYTE;
	TAP				: BYTE:=4;	   (* Consecutive checks filter *)
	INITEV			: BOOL:= TRUE; (* Generate init OK event *)
	IN_EMIN			: INT :=-2000; (* Low error limit *)
	IN_WMIN			: INT := -550; (* Low warning value *)
	IN_WMAX			: INT :=  900; (* High warning value *)
	IN_EMAX			: INT := 8500; (* High error limit *)
	ERR_MIN_SHORT	: BOOL:= TRUE; (* TRUE  ==> EMIN=Short        , EMAX=Disconnected
									  FALSE ==> EMIN=Disconnected , EMAX=Short 		 *)
	(* Physical input *)
	IN			: INT;
END_VAR
VAR_OUTPUT
	WRN			: BOOL;	(* Value in warning range *)
	ERR			: BOOL;	(* Value error *)
	HI			: INT;	(* Highest value - cleared by Stat_Reset() action *)
	AVG			: INT; 	(* Average value - updated by Mean() action, cleared by Mean_Reset() action *)
	LOW			: INT;	(* Lowest value  - cleared by Stat_Reset() action *)

	Status_Log	: WORD;
	Status_Vis	: DWORD;
END_VAR
VAR
	cnt			: BYTE;
	event		: BYTE := 0;	(* 0: monitoring a generic, 1: monitoring an error, 2: monitoring a warning *)
	asum		: DINT;
	acnt		: WORD;
END_VAR
(* Check probe value limits *)
IF IN<=IN_EMIN OR IN>=IN_EMAX THEN
	IF NOT ERR THEN
		IF event <> ErrorEv THEN
			cnt := 1;
			event := ErrorEv;
		ELSE
			cnt:=cnt+1;
		END_IF

		IF cnt>TAP THEN
			cnt:=0;
			ERR:=TRUE; WRN:=FALSE;
			IF ( ERR_MIN_SHORT=TRUE  AND IN<=IN_EMIN ) OR ( ERR_MIN_SHORT=FALSE AND IN>=IN_EMAX ) THEN
				LogEv(EL_Alarm,EO_TPV,ID,5,INT_TO_STRING(IN));
			ELSE
				LogEv(EL_Alarm,EO_TPV,ID,4,INT_TO_STRING(IN));
			END_IF
		END_IF
	END_IF
ELSIF IN<=IN_WMIN OR IN>=IN_WMAX THEN
	IF NOT WRN THEN
		IF event <> WarningEv THEN
			cnt := 1;
			event := WarningEv;
		ELSE
			cnt:=cnt+1;
		END_IF

		IF cnt>TAP THEN
			cnt:=0;
			ERR:=FALSE; WRN:=TRUE;
			LogEv(EL_Wrn,EO_TPV,ID,SEL(IN<=IN_WMIN,3,2),INT_TO_STRING(IN));
		END_IF
	END_IF
ELSE
	IF INITEV OR WRN OR ERR THEN
		IF event <> NormalEv THEN
			cnt := 1;
			event := NormalEv;
		ELSE
			cnt:=cnt+1;
		END_IF

		IF cnt>TAP THEN
			cnt:=0;
			INITEV:=FALSE; ERR:=FALSE; WRN:=FALSE;
			LogEv(EL_Log,EO_TPV,ID,1,'Probe_OK');
		END_IF
	END_IF
END_IF


(*
(* Average value *)
IF acnt>=500 THEN
	Mean();
	asum := asum - AVG;
	acnt := acnt - 1;
END_IF

asum := asum + IN;
acnt := acnt + 1;
*)

AVG := IN;



(* Statistics values *)
IF IN<LOW THEN LOW:=IN; END_IF
IF IN>HI  THEN HI :=IN; END_IF



(* Status Log *)
IF ERR THEN	Status_Log := 2; Status_Vis := COLOR_RED;
ELSIF WRN THEN Status_Log := 1;	Status_Vis := COLOR_YELLOW;
ELSE Status_Log := 0; Status_Vis := COLOR_GREEN;
END_IF
END_FUNCTION_BLOCK
ACTION AddLogData:
Logger.s1:=INSERT('&TPV=',BYTE_TO_STRING(ID),4);
IF ID<10 THEN Logger.s1:=INSERT(Logger.s1,'0',4); END_IF
(*
Mean();
*)
Logger.s1:=CONCAT(Logger.s1,INT_TO_STRING(AVG));		Logger.s1:=CONCAT(Logger.s1,';');

Logger.s1:=CONCAT(Logger.s1,WORD_TO_STRING(Status_Log));
ADDSTRING(ADR(Logger.TData), ADR(Logger.s1), Logger.TLen);
END_ACTION
ACTION Mean:
AVG := DINT_TO_INT(asum/acnt);
END_ACTION
ACTION Mean_Reset:
AVG:=IN;
asum:=IN;
acnt:=1;
END_ACTION
ACTION Stat_Reset:
HI:=IN;
LOW:=IN;
END_ACTION

(* POU Plant_Objects/obj_VRD_02, ST *)
FUNCTION_BLOCK obj_VRD_02
(* === VALVOLA RIPARTITORE ===
  VERSIONE 01 REALIZZATA DA MORENO E TESTATA SU IMPIANTO SAN FELICE ID 012 CLV

			02   - 	Introdotto possibilità di impstare il set point in Automatico ( da curva Cliamtica ) o da remoto ( set Point
				 	impostato fuori dalla FB per dare un Set Point Fisso.
				 -	Introdotto Temperatura di Controllo Curva climatica con paramentro di ingresso delle FB 



*)
VAR CONSTANT
	Chk_CntSecAlarm	: INT := 900;	(* 900s = 15 minutes -> Observation itme *)
END_VAR

VAR_INPUT
	(* Settings *)
	ID				: BYTE;
	(* Controls *)
	RUN  			: BOOL;					(* Control input *)
	ReducedRange	: BOOL := FALSE;		(* If true output value is among 2 and 10V, otherwise 0-10V *)

	(* Physical inputs *)
	TEMP 			: INT;		(* Input temperature from sensor *)
	STATUS 			: WORD;		(* Input position from valve *)

	InitOK			: BOOL;
	Alarm1			: BOOL;
	Alarm2			: BOOL;
	Warning			: BOOL;

	Ctrl_Init		: BOOL;
	Ctrl_SetPoint	: INT;
	Ctrl_SetPointNew: INT := 0;
	Delta_SetPoint	: INT;
	Ctrl_Err		: INT;			(* Current error *)
	Ctrl_Err0		: INT; 			(* Previous error *)
	Ctrl_Accel		: REAL;			(* Derivate of error *)
	Ctrl_AccelGate  : INT:=1;		(* Derivate gate *)
	Ctrl_AccelTmr	: WORD;
	Ctrl_SetPointGate: INT := 5;	(* Setpoint gate - 0.5°C *)
	Ctrl_Out		: REAL;

	Chk_Err			: INT;
	Chk_Cnt			: INT;
	Chk_CntAlarm	: INT:=240; 		(* Check error trigger 120s *)

	(* Status *)
	Log_AvgTemp		: AVERAGE_T;
	Status_Log		: BYTE;
	Status_Vis 		: DWORD;

	(* Feedback *)
	fFeedback		: BOOL;			(* TRUE: Feedback available, FALSE: Feedback not available *)

	OffsetBoost: INT;

	ComandoManuale:BOOL:=FALSE;
	RiferimentoManuale:INT;

	TempControlloCC:INT;

	AbilitaSetPointManuale: BOOL:=FALSE;
	SetPointManuale: INT:=400;


END_VAR
VAR_IN_OUT
	CLIM		: typ_Clima;
END_VAR
VAR_OUTPUT
	(* Physical outputs *)
	OUT			: WORD;
END_VAR
VAR
	Curve		: CHARCURVE;
	Curve_Err	: BYTE;

	aTemp		: ARRAY [1..20] OF INT;
	meanTemp	: INT;
	sum			: INT := 0;
	Tmr			: TON := (PT:=T#1s);
	index		: BYTE;
	i			: BYTE;
	fCtrl_Err	: BOOL;		(* TRUE: Ctrl_Err>0, FALSE: Ctrl_Err<0 *)

	SetPoint: INT;
END_VAR

VAR_INPUT RETAIN
	Ctrl_ErrGate	: INT:=5;		(* Error gate *)
	Chk_ErrGate		: INT:=3200; 		(* Check error gate *)
	Ctrl_Kp			: REAL:=2;(*1;*)		(* Proportional factor *)
	Ctrl_Kd			: REAL:=10;(*100;*)  	(* Derivative factor *)

	Local_VRD_TAlarm: INT;

END_VAR
(* Check initialization *)
(*IF NOT InitOK THEN Init(); END_IF*)

(* Check max temperature *)
IF TEMP>Local_VRD_TAlarm THEN
	IF NOT Alarm1 THEN
		Alarm1:=TRUE;
		LogEv(EL_AlarmStop,EO_VRD,ID,3,'VRD_Overtemperature');
	END_IF
ELSE
	Alarm1:=FALSE;
END_IF

(* Check climatic setup *)
IF NOT CLIM.InitOK THEN	DefaultClim(); END_IF;
(* Calculate Setpoint *)
Curve(	IN:= TempControlloCC,	N:= 5, P:= CLIM.Points,			(* Given the x value as input, the corresponding y value as output is returned, if it matches the crve designed by array of points *)
		OUT=> Ctrl_SetPointNew, ERR=> Curve_Err );


(*IF Curve_Err>0 OR Ctrl_SetPoint>Local_VRD_TAlarm THEN*)
IF  Ctrl_SetPoint>Local_VRD_TAlarm THEN
	Ctrl_SetPoint:=Local_VRD_TAlarm;
	IF NOT Warning THEN
		Warning:=TRUE;
		LogEv(EL_Wrn,EO_VRD,ID,2,'VRD_Climatic_Error');
	END_IF
ELSE
	Delta_SetPoint := ABS(Ctrl_SetPoint - Ctrl_SetPointNew);
	IF Delta_SetPoint>Ctrl_SetPointGate THEN Ctrl_SetPoint := Ctrl_SetPointNew; END_IF

	Warning:=FALSE;
END_IF



(* Scelta del set point della VRD o vien preso dalla curva cliamtica o da un riferimento esterno *)
IF AbilitaSetPointManuale THEN
	SetPoint:=SetPointManuale;
ELSE
	SetPoint:=Ctrl_SetPointNew;
END_IF




SetPoint:=SetPoint+OffsetBoost;    (* Aggiungo l'eventuale Offset di Boost al Set point da passare alla regolatore *)


(* Execute control loop [T=500ms] *)
IF RUN AND (NOT Alarm1) THEN
	(* Calculate error *)
	Ctrl_Err:=SetPoint-TEMP;
	(* Init/restart operations *)
	IF NOT Ctrl_Init THEN
		Ctrl_Accel:=0;
		Ctrl_AccelTmr:=0;
		Ctrl_Err0:=Ctrl_Err;
		Ctrl_Out:=5000;
		Ctrl_Init:=TRUE;
	END_IF
	(* Calculate acceleration *)
	IF ABS(Ctrl_Err-Ctrl_Err0)>Ctrl_AccelGate OR Ctrl_AccelTmr>20 THEN
		Ctrl_Accel:=INT_TO_REAL(Ctrl_Err-Ctrl_Err0)/WORD_TO_REAL(1+Ctrl_AccelTmr);
		Ctrl_AccelTmr:=0;
		Ctrl_Err0:=Ctrl_Err;
	ELSE
		Ctrl_AccelTmr:=Ctrl_AccelTmr+1;
	END_IF

	(* Gate error *)
	IF ABS(Ctrl_Err)>Ctrl_ErrGate THEN
		(* Control loop *)
		Ctrl_Out:=Ctrl_Out+(Ctrl_Kp*Ctrl_Err)+(Ctrl_Kd*Ctrl_Accel);
	END_IF

	(* Limiter and Output *)

	IF NOT ComandoManuale THEN
		Ctrl_Out:=LIMIT(0,Ctrl_Out,32766);
	ELSE
		RiferimentoManuale:=LIMIT(0,REAL_TO_INT(RiferimentoManuale),100); 	(* il comando è espresso in percentuale *)
		Ctrl_Out:=RiferimentoManuale*327; 									(* il comando è espresso in percentuale *)
	END_IF

	OUT:=REAL_TO_WORD(Ctrl_Out);

ELSE
	Ctrl_Init:=FALSE;
	OUT:=0;
END_IF

(* If there is an hardware feedback (such as 0-10V, potentiometer, ...) check it otherwise try to rebuild it *)
IF fFeedback THEN CheckFeedback();
ELSE BuildFeedback();
END_IF

(* Status temp *)
Log_AvgTemp(IN:=Temp);
(* Lamp.UpdateStatus(obj_Status := Status_Log); *)

(* Status color *)
   IF Alarm1 OR Alarm2 THEN Status_Log:=2; Status_Vis:=16#2020F0;
ELSIF Warning          THEN Status_Log:=1; Status_Vis:=16#20F0F0;
                       ELSE Status_Log:=0; Status_Vis:=SEL(RUN,16#006000,16#20F020);
END_IF
END_FUNCTION_BLOCK
ACTION AddLogData:
Logger.s1:=INSERT('&VRD=',BYTE_TO_STRING(ID),4);
IF ID<10 THEN Logger.s1:=INSERT(Logger.s1,'0',4); END_IF

Logger.s1:=CONCAT(Logger.s1,INT_TO_STRING(SetPoint));
Logger.s1:=CONCAT(Logger.s1,';');
Logger.s1:=CONCAT(Logger.s1,WORD_TO_STRING(OUT/327));
Logger.s1:=CONCAT(Logger.s1,';');

IF fFeedback THEN Logger.s1:=CONCAT(Logger.s1,WORD_TO_STRING(STATUS/327));
ELSE Logger.s1:=CONCAT(Logger.s1,'0');	(* Bypass *)
END_IF

Logger.s1:=CONCAT(Logger.s1,';');

Logger.s1:=CONCAT(Logger.s1,WORD_TO_STRING(Status_Log));
ADDSTRING(ADR(Logger.TData), ADR(Logger.s1), Logger.TLen);
END_ACTION
ACTION BuildFeedback:
(* Comparison is taken between actual temperature vs windowed mean value of last 20 temperature
   (check is carried out every second)	*)
IF RUN AND (NOT Alarm1) THEN

	IF Ctrl_Err>0 THEN
		IF NOT fCtrl_Err THEN index := 0; END_IF
		fCtrl_Err := TRUE;
	ELSE
		IF fCtrl_Err THEN index := 0; END_IF
		fCtrl_Err := FALSE;
	END_IF

	(* Temperature is lower than setpoint -->> Should increase *)
	Tmr(IN:=NOT Tmr.Q);

	IF Tmr.Q THEN

		IF index<21 THEN
			(* Fullfil temperature array *)
			aTemp[index] := TEMP;
			index := index + 1;

			IF index=20 THEN
				FOR i:=1 TO 20 BY 1 DO sum := sum + aTemp[i]; END_FOR
			END_IF
		ELSE
			(* Calculate mean value *)
			meanTemp := sum/20;

			IF (fCtrl_Err AND TEMP<meanTemp) OR (NOT fCtrl_Err AND TEMP>meanTemp) THEN

				IF Chk_Cnt>Chk_CntSecAlarm THEN
					IF NOT Alarm2 THEN
						Alarm2:=TRUE;
						LogEv(EL_Alarm,EO_VRD,ID,4,'VRD_Position_Error');
					END_IF
				ELSE
					Chk_Cnt := Chk_Cnt+1;
				END_IF

			ELSE
				(* Reset counter and alarm flag *)
				Chk_Cnt:=0;
				Alarm2:=FALSE;
			END_IF

			sum := 0;	(* Reset sum counter *)

			(* Shift array removing oldest value *)
			FOR i:=1 TO 20 BY 1 DO
				aTemp[i-1] := aTemp[i];
				sum := sum + aTemp[i];
			END_FOR

			aTemp[20] := TEMP;			(* Last temperature value is new one *)
			sum := sum + aTemp[20];		(* Update sum *)
		END_IF
	END_IF
END_IF
END_ACTION
ACTION CheckFeedback:
(* Calculate position error according to feedback *)
IF ReducedRange THEN
(* SETPOINT[2..10V]-STATUS[0..10V] *)
	IF OUT<=6553 THEN Chk_Err:=0; ELSE Chk_Err:=(OUT-6553)/262; END_IF
	Chk_Err:=(Chk_Err-STATUS)/327;
ELSE
(* SETPOINT[0..10V]-STATUS[0..10V] *)
	Chk_Err := OUT - STATUS;
END_IF

(* Check position error *)
IF ( ABS(Chk_Err)>Chk_ErrGate ) THEN
	IF Chk_Cnt>Chk_CntAlarm THEN
		IF NOT Alarm2 THEN
			Alarm2:=TRUE;
			LogEv(EL_Alarm,EO_VRD,ID,4,'VRD_Position_Error');
		END_IF
	ELSE
		Chk_Cnt:=Chk_Cnt+1;
	END_IF
ELSE
	Chk_Cnt:=0;
	Alarm2:=FALSE;
END_IF
END_ACTION
ACTION DefaultClim:
(*CLIM.Points[0].X:=-300; CLIM.Points[0].Y:=400;
CLIM.Points[1].X:=-50;  CLIM.Points[1].Y:=400;
CLIM.Points[2].X:= 200; CLIM.Points[2].Y:=200;
CLIM.Points[3].X:= 300; CLIM.Points[3].Y:=200;
CLIM.Points[4].X:= 500; CLIM.Points[4].Y:=200;*)
IF CLIM.Points[0].X=0 THEN

CLIM.Points[0].X:=-50; CLIM.Points[0].Y:=750;
CLIM.Points[1].X:=0 ; CLIM.Points[1].Y:=700;
CLIM.Points[2].X:= 100;  CLIM.Points[2].Y:=600;
CLIM.Points[3].X:= 150; CLIM.Points[3].Y:=500;
CLIM.Points[4].X:= 200; CLIM.Points[4].Y:=350;

END_IF


CLIM.InitOK:=TRUE;
LogEv(EL_Wrn,EO_VRD,ID,1,'Climatic_Default');
END_ACTION
ACTION Init:
(* End initialization *)
InitOK:=TRUE;
END_ACTION

(* POU Utils Functions/PLANT_STATUS, ST *)
FUNCTION_BLOCK PLANT_STATUS
VAR_INPUT
	obj_Status		:	WORD;
END_VAR
VAR_OUTPUT
END_VAR
VAR
	PLANT_STATUS	:	WORD;

	Pwm				:	TON := (PT:=T#1s);
END_VAR
CASE plant_Status OF

	0:	(* Plant OK - Everything works well *)
		(*Pwm(IN:=FALSE);	*)						(* Stop timer if running *)
		LAMP_AL := FALSE;						(* Keep the lamp switched off *)

	(*1:	(* Plant in warning *)
		Pwm(IN:= NOT(Pwm.Q));

		IF Pwm.Q THEN
			LAMP_AL := NOT LAMP_AL;				(* Toggle output *)
		END_IF*)

	2:	(* Plant in alarm *)
		(*Pwm(IN:=FALSE);	*)						(* Stop timer if running *)
		LAMP_AL	:= TRUE;						(* Keep the lamp switched on *)

END_CASE

plant_Status := 0;		(* Reset plant status *)
END_FUNCTION_BLOCK
ACTION UpdateStatus:
IF plant_Status = 2 THEN

	RETURN;					(* If plant already in alarm condition do nothing *)

ELSE

		IF obj_Status <> 0 THEN
			plant_Status := obj_Status;			(* If plant in warning/normal condition and current object in alarm, update plant status *)
		END_IF
END_IF
END_ACTION

(* POU PLC_WDT, ST *)
FUNCTION PLC_WDT: DWORD VAR_INPUT dwEvent: DWORD; dwFilter: DWORD; dwOwner: DWORD; END_VAR
LogEv(EL_AlarmStop,EO_SYS,1,10,'Watchdog');
END_FUNCTION

(* POU Utils Functions/RAW16TOHEXSTR, ST *)
FUNCTION RAW16TOHEXSTR : STRING(128)
VAR_INPUT
	pData: POINTER TO BYTE;
	DataLen: BYTE;
END_VAR
VAR
	pt: POINTER TO BYTE;
	xl: BYTE;
END_VAR
pt:=ADR(RAW16TOHEXSTR);
xl:=0;

WHILE DataLen>0 AND xl<120 DO

	pData:=pData+1;

	pt^ := (pData^ / 16#10) + 48 + (((pData^ / 16#10)/10)*7);
	pt:=pt+1;
	pt^ := (pData^ AND 16#0F)  + 48 + (((pData^ AND 16#0F)/10)*7);
	pt:=pt+1;

	pData:=pData-1;

	pt^ := (pData^ / 16#10) + 48 + (((pData^ / 16#10)/10)*7);
	pt:=pt+1;
	pt^ := (pData^ AND 16#0F)  + 48 + (((pData^ AND 16#0F)/10)*7);
	pt:=pt+1;

	xl:=xl+4;

	DataLen:=DataLen-2;
	pData:=pData+2;

END_WHILE

pt^:=0;
END_FUNCTION

(* POU Utils Functions/RAWTOHEXSTR, ST *)
FUNCTION RAWTOHEXSTR : STRING(128)
VAR_INPUT
	pData: POINTER TO BYTE;
	DataLen: BYTE;
END_VAR
VAR
	pt: POINTER TO BYTE;
	xl: BYTE;
END_VAR
pt:=ADR(RAWTOHEXSTR);

xl:=2;

WHILE DataLen>0 AND xl<128 DO

	pt^ := (pData^ / 16#10) + 48 + (((pData^ / 16#10)/10)*7);
	pt:=pt+1;
	pt^ := (pData^ AND 16#0F)  + 48 + (((pData^ AND 16#0F)/10)*7);
	pt:=pt+1;

	xl:=xl+2;

	DataLen:=DataLen-1;
	pData:=pData+1;

END_WHILE

pt^:=0;
END_FUNCTION

(* POU Utils/RTC_Update, ST *)
FUNCTION RTC_Update : BOOL
VAR
	T: DT;
	TS: STRING;
	TS2: STRING;
	Hour: BYTE;
	Minute: BYTE;
END_VAR
(* Get RTC time *)
T:=SysRtcGetTime(TRUE);
Sys.Time_CT_DT:=T;
(* Calculate variables *)
TS:=DT_TO_STRING(T);
Sys.Time_LogString:=DELETE(STR:=TS, LEN:=3, POS:=1);
TS2:=MID(STR:=TS, LEN:=4, POS:= 4); Sys.Time_Year 	:=STRING_TO_WORD(TS2);
TS2:=MID(STR:=TS, LEN:=2, POS:= 9); Sys.Time_Month	:=STRING_TO_BYTE(TS2);
TS2:=MID(STR:=TS, LEN:=2, POS:=12); Sys.Time_Day  	:=STRING_TO_BYTE(TS2);
Sys.Time_CT_Day:=(32*(Sys.Time_Month-1)+Sys.Time_Day-1);
TS2:=MID(STR:=TS, LEN:=2, POS:=15); Hour			:=STRING_TO_BYTE(TS2);
TS2:=MID(STR:=TS, LEN:=2, POS:=18); Minute		 	:=STRING_TO_BYTE(TS2);
Sys.Time_Hour := Hour;
Sys.Time_Minute := Minute;
Sys.Time_CT_Quarter:=Hour*4+(Minute/15);
END_FUNCTION

(* POU Utils Functions/SHIFT_ARRAY, ST *)
FUNCTION SHIFT_ARRAY : BOOL
VAR_INPUT
	pData	:	POINTER TO ARRAY [1..2] OF WORD;
	Size	:	BYTE;
END_VAR
VAR
	pNew	:	POINTER TO WORD;
	i		:	BYTE;
END_VAR
(* Shift right *)
FOR i:=1 TO (Size-1) BY 1 DO

	(*pNew := pData + 1;*)
	pData^[i] := pData^[i+1];
	(*pData := pData + 1;*)

END_FOR
END_FUNCTION

(* Visualisation PLC_VISU
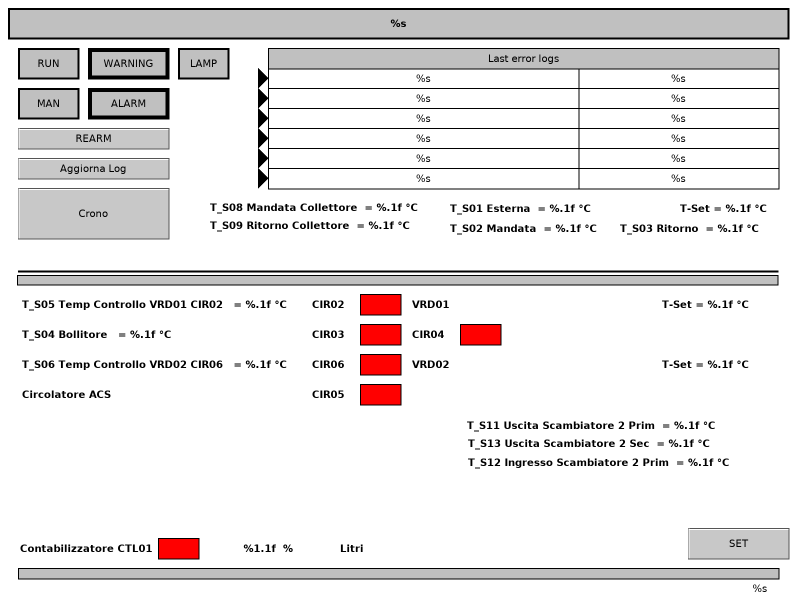
rectangle at (10,10)-(791,41): text "%s"; shows .Plant_NAME
rectangle at (530,580)-(771,601): text "%s"; shows Sys.Time_LogString
rounded rectangle at (20,50)-(81,81): text "RUN"; alarm colour if NOT Mode_Manual; runs INTERN ASSIGN Mode_Manual:=(FALSE)
rounded rectangle at (20,90)-(81,121): text "MAN"; alarm colour if Mode_Manual; runs INTERN ASSIGN Mode_Manual:=(TRUE)
rectangle at (580,70)-(781,91): text "%s"; shows Sys.LastLogs_Msg[0]
polygon at (260,170)-(270,190): invisible if Sys.LastLogs_Idx<>0
rectangle at (580,90)-(781,111): text "%s"; shows Sys.LastLogs_Msg[1]
polygon at (260,70)-(270,90): invisible if Sys.LastLogs_Idx<>1
rectangle at (580,110)-(781,131): text "%s"; shows Sys.LastLogs_Msg[2]
polygon at (260,90)-(270,110): invisible if Sys.LastLogs_Idx<>2
rectangle at (580,130)-(781,151): text "%s"; shows Sys.LastLogs_Msg[3]
polygon at (260,110)-(270,130): invisible if Sys.LastLogs_Idx<>3
rectangle at (580,150)-(781,171): text "%s"; shows Sys.LastLogs_Msg[4]
polygon at (260,130)-(270,150): invisible if Sys.LastLogs_Idx<>4
rectangle at (580,170)-(781,191): text "%s"; shows Sys.LastLogs_Msg[5]
polygon at (260,150)-(270,170): invisible if Sys.LastLogs_Idx<>5
rectangle at (270,70)-(581,91): text "%s"; shows Sys.LastLogs_Dat[0]
rectangle at (270,90)-(581,111): text "%s"; shows Sys.LastLogs_Dat[1]
rectangle at (270,110)-(581,131): text "%s"; shows Sys.LastLogs_Dat[2]
rectangle at (270,130)-(581,151): text "%s"; shows Sys.LastLogs_Dat[3]
rectangle at (270,150)-(581,171): text "%s"; shows Sys.LastLogs_Dat[4]
rectangle at (270,170)-(581,191): text "%s"; shows Sys.LastLogs_Dat[5]
rectangle at (90,90)-(171,121): text "ALARM"; alarm colour if Sys.Alarm; runs INTERN ASSIGN Mode_Manual:=(FALSE)
rectangle at (90,50)-(171,81): text "WARNING"; alarm colour if Sys.Warning; runs INTERN ASSIGN Mode_Manual:=(TRUE)
button at (20,130)-(171,151): text "REARM"; runs INTERN ASSIGN Sys.Alarm:=(FALSE);INTERN ASSIGN Sys.Warning:=(FALSE)
rectangle at (270,50)-(781,71): text "Last error logs"
rounded rectangle at (180,50)-(231,81): text "LAMP"; alarm colour if LAMP_AL
rectangle at (450,200)-(661,221): text "T_S01 Esterna  = %.1f °C"; shows INT_TO_REAL(.TPV01.AVG)/10
rectangle at (450,220)-(661,241): text "T_S02 Mandata  = %.1f °C"; shows INT_TO_REAL(.TPV02.AVG)/10
rectangle at (620,220)-(771,241): text "T_S03 Ritorno  = %.1f °C"; shows INT_TO_REAL(.TPV03.IN)/10
rectangle at (22,326)-(233,347): text "T_S04 Bollitore   = %.1f °C"; shows INT_TO_REAL(.TPV04.IN)/10
rectangle at (22,296)-(313,317): text "T_S05 Temp Controllo VRD01 CIR02   = %.1f °C"; shows INT_TO_REAL(.TPV05.IN)/10
rectangle at (22,356)-(303,377): text "T_S06 Temp Controllo VRD02 CIR06   = %.1f °C"; shows INT_TO_REAL(.TPV06.IN)/10
button at (20,160)-(171,181): text "Aggiorna Log"; taps PLC_PRG.HMI_AggiornaLog
button at (20,190)-(171,241): text "Crono"; opens VIS_CHONOEDITOR
rectangle at (680,200)-(781,221): text "T-Set = %.1f °C"; shows INT_TO_REAL(.CAL01.SetPointCaldaia)/10
rectangle at (312,296)-(363,317): text "CIR02"
rectangle at (412,296)-(463,317): text "VRD01"
rectangle at (312,326)-(363,347): text "CIR03"
rectangle at (412,326)-(463,347): text "CIR04"
rectangle at (312,386)-(363,407): text "CIR05"
rectangle at (312,356)-(363,377): text "CIR06"
rectangle at (412,356)-(463,377): text "VRD02"
rectangle at (20,540)-(181,561): text "Contabilizzatore CTL01"; shows INT_TO_REAL(.TPV06.IN)/10)
rectangle at (160,540)-(201,561): alarm colour if .CTL01.CTL_ST
rectangle at (210,540)-(331,561): text "%1.1f  %"; shows DINT_TO_REAL(.CTL01.COUNT)/10
button at (690,530)-(791,561): text "SET"; opens VIS_SET
rectangle at (340,540)-(381,561): text "Litri"; shows INT_TO_REAL(.TPV06.IN)/10)
rectangle at (362,296)-(403,317): alarm colour if .CIR02_ST
rectangle at (362,326)-(403,347): alarm colour if .CIR03_ST
rectangle at (362,356)-(403,377): alarm colour if .CIR06_ST
rectangle at (462,326)-(503,347): alarm colour if .CIR04_ST
rectangle at (362,386)-(403,407): alarm colour if .CIR05_ST
rectangle at (22,386)-(303,407): text "Circolatore ACS"; shows INT_TO_REAL(.TPV06.IN)/10
rectangle at (662,296)-(763,317): text "T-Set = %.1f °C"; shows INT_TO_REAL(.VRD01.Ctrl_SetPoint)/10
rectangle at (662,356)-(763,377): text "T-Set = %.1f °C"; shows INT_TO_REAL(.VRD02.Ctrl_SetPoint)/10
rectangle at (210,199)-(430,220): text "T_S08 Mandata Collettore  = %.1f °C"; shows INT_TO_REAL(.TPV08.AVG)/10
rectangle at (210,217)-(421,238): text "T_S09 Ritorno Collettore  = %.1f °C"; shows INT_TO_REAL(.TPV09.AVG)/10
rectangle at (467,417)-(733,438): text "T_S11 Uscita Scambiatore 2 Prim  = %.1f °C"; shows INT_TO_REAL(.TPV11.AVG)/10
rectangle at (468,435)-(759,456): text "T_S13 Uscita Scambiatore 2 Sec  = %.1f °C"; shows INT_TO_REAL(.TPV13.AVG)/10
rectangle at (468,454)-(759,475): text "T_S12 Ingresso Scambiatore 2 Prim  = %.1f °C"; shows INT_TO_REAL(.TPV12.AVG)/10
3 more shapes without text or variables
4 elements of other kinds (tables, trends, ...) not read
*)

(* Visualisation VIS_CHONOEDITOR
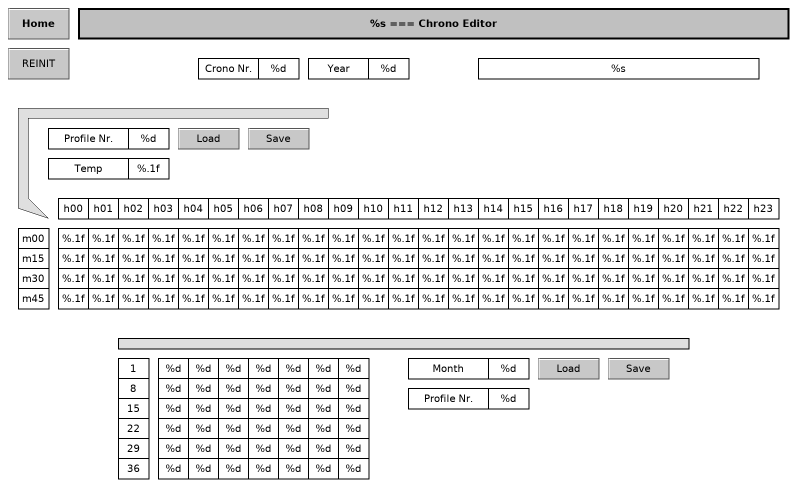
rectangle at (200,60)-(261,81): text "Crono Nr."
rectangle at (260,60)-(301,81): text "%d"; shows CronEd.CN_Sel; alarm colour if CronEd.CN_Sel<>CronEd.CN_Act; editable 1..6
rectangle at (50,130)-(131,151): text "Profile Nr."
rectangle at (130,130)-(171,151): text "%d"; shows CronEd.PR_Sel; alarm colour if CronEd.PR_Sel<>CronEd.PR_Act; editable 1..10
rectangle at (50,160)-(131,181): text "Temp"
rectangle at (130,160)-(171,181): text "%.1f"; shows CronEd.PR_TT; editable
button at (180,130)-(241,151): text "Load"; toggles CronEd.PR_Load
button at (250,130)-(311,151): text "Save"; toggles CronEd.PR_Save
rectangle at (20,230)-(51,251): text "m00"
rectangle at (20,250)-(51,271): text "m15"
rectangle at (20,270)-(51,291): text "m30"
rectangle at (20,290)-(51,311): text "m45"
rectangle at (80,10)-(791,41): text "%s === Chrono Editor"; shows .Plant_NAME
button at (10,10)-(71,41): text "Home"; opens PLC_VISU
rounded rectangle at (60,230)-(91,251): text "%.1f"; shows WORD_TO_REAL(CronEd.PR.Setpoint[0])/10; runs INTERN ASSIGN CronEd.PR.Setpoint[0]:=(REAL_TO_WORD(CronEd.PR_TT*10))
rounded rectangle at (60,250)-(91,271): text "%.1f"; shows WORD_TO_REAL(CronEd.PR.Setpoint[1])/10; runs INTERN ASSIGN CronEd.PR.Setpoint[1]:=(REAL_TO_WORD(CronEd.PR_TT*10))
rounded rectangle at (60,270)-(91,291): text "%.1f"; shows WORD_TO_REAL(CronEd.PR.Setpoint[2])/10; runs INTERN ASSIGN CronEd.PR.Setpoint[2]:=(REAL_TO_WORD(CronEd.PR_TT*10))
rounded rectangle at (60,290)-(91,311): text "%.1f"; shows WORD_TO_REAL(CronEd.PR.Setpoint[3])/10; runs INTERN ASSIGN CronEd.PR.Setpoint[3]:=(REAL_TO_WORD(CronEd.PR_TT*10))
rectangle at (60,200)-(91,221): text "h00"; runs INTERN ASSIGN CronEd.PR.Setpoint[0]:=(REAL_TO_WORD(CronEd.PR_TT*10));INTERN ASSIGN CronEd.PR.Setpoint[1]:=(REAL_TO_WORD(CronEd.PR_TT*10));INTERN ASSIGN CronEd.PR.Setpoint[2]:=(REAL_TO_WORD(CronEd.PR_TT*10));INTERN ASSIGN CronEd.PR.Setpoint[3]:=(REAL_TO_WORD(CronEd.PR_TT*10))
rounded rectangle at (90,230)-(121,251): text "%.1f"; shows WORD_TO_REAL(CronEd.PR.Setpoint[4])/10; runs INTERN ASSIGN CronEd.PR.Setpoint[4]:=(REAL_TO_WORD(CronEd.PR_TT*10))
rounded rectangle at (90,250)-(121,271): text "%.1f"; shows WORD_TO_REAL(CronEd.PR.Setpoint[5])/10; runs INTERN ASSIGN CronEd.PR.Setpoint[5]:=(REAL_TO_WORD(CronEd.PR_TT*10))
rounded rectangle at (90,270)-(121,291): text "%.1f"; shows WORD_TO_REAL(CronEd.PR.Setpoint[6])/10; runs INTERN ASSIGN CronEd.PR.Setpoint[6]:=(REAL_TO_WORD(CronEd.PR_TT*10))
rounded rectangle at (90,290)-(121,311): text "%.1f"; shows WORD_TO_REAL(CronEd.PR.Setpoint[7])/10; runs INTERN ASSIGN CronEd.PR.Setpoint[7]:=(REAL_TO_WORD(CronEd.PR_TT*10))
rectangle at (90,200)-(121,221): text "h01"; runs INTERN ASSIGN CronEd.PR.Setpoint[4]:=(REAL_TO_WORD(CronEd.PR_TT*10));INTERN ASSIGN CronEd.PR.Setpoint[5]:=(REAL_TO_WORD(CronEd.PR_TT*10));INTERN ASSIGN CronEd.PR.Setpoint[6]:=(REAL_TO_WORD(CronEd.PR_TT*10));INTERN ASSIGN CronEd.PR.Setpoint[7]:=(REAL_TO_WORD(CronEd.PR_TT*10))
rounded rectangle at (120,230)-(151,251): text "%.1f"; shows WORD_TO_REAL(CronEd.PR.Setpoint[8])/10; runs INTERN ASSIGN CronEd.PR.Setpoint[8]:=(REAL_TO_WORD(CronEd.PR_TT*10))
rounded rectangle at (120,250)-(151,271): text "%.1f"; shows WORD_TO_REAL(CronEd.PR.Setpoint[9])/10; runs INTERN ASSIGN CronEd.PR.Setpoint[9]:=(REAL_TO_WORD(CronEd.PR_TT*10))
rounded rectangle at (120,270)-(151,291): text "%.1f"; shows WORD_TO_REAL(CronEd.PR.Setpoint[10])/10; runs INTERN ASSIGN CronEd.PR.Setpoint[10]:=(REAL_TO_WORD(CronEd.PR_TT*10))
rounded rectangle at (120,290)-(151,311): text "%.1f"; shows WORD_TO_REAL(CronEd.PR.Setpoint[11])/10; runs INTERN ASSIGN CronEd.PR.Setpoint[11]:=(REAL_TO_WORD(CronEd.PR_TT*10))
rectangle at (120,200)-(151,221): text "h02"; runs INTERN ASSIGN CronEd.PR.Setpoint[8]:=(REAL_TO_WORD(CronEd.PR_TT*10));INTERN ASSIGN CronEd.PR.Setpoint[9]:=(REAL_TO_WORD(CronEd.PR_TT*10));INTERN ASSIGN CronEd.PR.Setpoint[10]:=(REAL_TO_WORD(CronEd.PR_TT*10));INTERN ASSIGN CronEd.PR.Setpoint[11]:=(REAL_TO_WORD(CronEd.PR_TT*10))
rounded rectangle at (150,230)-(181,251): text "%.1f"; shows WORD_TO_REAL(CronEd.PR.Setpoint[12])/10; runs INTERN ASSIGN CronEd.PR.Setpoint[12]:=(REAL_TO_WORD(CronEd.PR_TT*10))
rounded rectangle at (150,250)-(181,271): text "%.1f"; shows WORD_TO_REAL(CronEd.PR.Setpoint[13])/10; runs INTERN ASSIGN CronEd.PR.Setpoint[13]:=(REAL_TO_WORD(CronEd.PR_TT*10))
rounded rectangle at (150,270)-(181,291): text "%.1f"; shows WORD_TO_REAL(CronEd.PR.Setpoint[14])/10; runs INTERN ASSIGN CronEd.PR.Setpoint[14]:=(REAL_TO_WORD(CronEd.PR_TT*10))
rounded rectangle at (150,290)-(181,311): text "%.1f"; shows WORD_TO_REAL(CronEd.PR.Setpoint[15])/10; runs INTERN ASSIGN CronEd.PR.Setpoint[15]:=(REAL_TO_WORD(CronEd.PR_TT*10))
rectangle at (150,200)-(181,221): text "h03"; runs INTERN ASSIGN CronEd.PR.Setpoint[15]:=(REAL_TO_WORD(CronEd.PR_TT*10));INTERN ASSIGN CronEd.PR.Setpoint[14]:=(REAL_TO_WORD(CronEd.PR_TT*10));INTERN ASSIGN CronEd.PR.Setpoint[13]:=(REAL_TO_WORD(CronEd.PR_TT*10));INTERN ASSIGN CronEd.PR.Setpoint[12]:=(REAL_TO_WORD(CronEd.PR_TT*10))
rounded rectangle at (180,230)-(211,251): text "%.1f"; shows WORD_TO_REAL(CronEd.PR.Setpoint[16])/10; runs INTERN ASSIGN CronEd.PR.Setpoint[16]:=(REAL_TO_WORD(CronEd.PR_TT*10))
rounded rectangle at (180,250)-(211,271): text "%.1f"; shows WORD_TO_REAL(CronEd.PR.Setpoint[17])/10; runs INTERN ASSIGN CronEd.PR.Setpoint[17]:=(REAL_TO_WORD(CronEd.PR_TT*10))
rounded rectangle at (180,270)-(211,291): text "%.1f"; shows WORD_TO_REAL(CronEd.PR.Setpoint[18])/10; runs INTERN ASSIGN CronEd.PR.Setpoint[18]:=(REAL_TO_WORD(CronEd.PR_TT*10))
rounded rectangle at (180,290)-(211,311): text "%.1f"; shows WORD_TO_REAL(CronEd.PR.Setpoint[19])/10; runs INTERN ASSIGN CronEd.PR.Setpoint[19]:=(REAL_TO_WORD(CronEd.PR_TT*10))
rectangle at (180,200)-(211,221): text "h04"; runs INTERN ASSIGN CronEd.PR.Setpoint[19]:=(REAL_TO_WORD(CronEd.PR_TT*10));INTERN ASSIGN CronEd.PR.Setpoint[18]:=(REAL_TO_WORD(CronEd.PR_TT*10));INTERN ASSIGN CronEd.PR.Setpoint[17]:=(REAL_TO_WORD(CronEd.PR_TT*10));INTERN ASSIGN CronEd.PR.Setpoint[16]:=(REAL_TO_WORD(CronEd.PR_TT*10))
rounded rectangle at (210,230)-(241,251): text "%.1f"; shows WORD_TO_REAL(CronEd.PR.Setpoint[20])/10; runs INTERN ASSIGN CronEd.PR.Setpoint[20]:=(REAL_TO_WORD(CronEd.PR_TT*10))
rounded rectangle at (210,250)-(241,271): text "%.1f"; shows WORD_TO_REAL(CronEd.PR.Setpoint[21])/10; runs INTERN ASSIGN CronEd.PR.Setpoint[21]:=(REAL_TO_WORD(CronEd.PR_TT*10))
rounded rectangle at (210,270)-(241,291): text "%.1f"; shows WORD_TO_REAL(CronEd.PR.Setpoint[22])/10; runs INTERN ASSIGN CronEd.PR.Setpoint[22]:=(REAL_TO_WORD(CronEd.PR_TT*10))
rounded rectangle at (210,290)-(241,311): text "%.1f"; shows WORD_TO_REAL(CronEd.PR.Setpoint[23])/10; runs INTERN ASSIGN CronEd.PR.Setpoint[23]:=(REAL_TO_WORD(CronEd.PR_TT*10))
rectangle at (210,200)-(241,221): text "h05"; runs INTERN ASSIGN CronEd.PR.Setpoint[23]:=(REAL_TO_WORD(CronEd.PR_TT*10));INTERN ASSIGN CronEd.PR.Setpoint[22]:=(REAL_TO_WORD(CronEd.PR_TT*10));INTERN ASSIGN CronEd.PR.Setpoint[21]:=(REAL_TO_WORD(CronEd.PR_TT*10));INTERN ASSIGN CronEd.PR.Setpoint[20]:=(REAL_TO_WORD(CronEd.PR_TT*10))
rounded rectangle at (240,230)-(271,251): text "%.1f"; shows WORD_TO_REAL(CronEd.PR.Setpoint[24])/10; runs INTERN ASSIGN CronEd.PR.Setpoint[24]:=(REAL_TO_WORD(CronEd.PR_TT*10))
rounded rectangle at (240,250)-(271,271): text "%.1f"; shows WORD_TO_REAL(CronEd.PR.Setpoint[25])/10; runs INTERN ASSIGN CronEd.PR.Setpoint[25]:=(REAL_TO_WORD(CronEd.PR_TT*10))
rounded rectangle at (240,270)-(271,291): text "%.1f"; shows WORD_TO_REAL(CronEd.PR.Setpoint[26])/10; runs INTERN ASSIGN CronEd.PR.Setpoint[26]:=(REAL_TO_WORD(CronEd.PR_TT*10))
rounded rectangle at (240,290)-(271,311): text "%.1f"; shows WORD_TO_REAL(CronEd.PR.Setpoint[27])/10; runs INTERN ASSIGN CronEd.PR.Setpoint[27]:=(REAL_TO_WORD(CronEd.PR_TT*10))
rectangle at (240,200)-(271,221): text "h06"; runs INTERN ASSIGN CronEd.PR.Setpoint[27]:=(REAL_TO_WORD(CronEd.PR_TT*10));INTERN ASSIGN CronEd.PR.Setpoint[26]:=(REAL_TO_WORD(CronEd.PR_TT*10));INTERN ASSIGN CronEd.PR.Setpoint[25]:=(REAL_TO_WORD(CronEd.PR_TT*10));INTERN ASSIGN CronEd.PR.Setpoint[24]:=(REAL_TO_WORD(CronEd.PR_TT*10))
rounded rectangle at (270,230)-(301,251): text "%.1f"; shows WORD_TO_REAL(CronEd.PR.Setpoint[28])/10; runs INTERN ASSIGN CronEd.PR.Setpoint[28]:=(REAL_TO_WORD(CronEd.PR_TT*10))
rounded rectangle at (270,250)-(301,271): text "%.1f"; shows WORD_TO_REAL(CronEd.PR.Setpoint[29])/10; runs INTERN ASSIGN CronEd.PR.Setpoint[29]:=(REAL_TO_WORD(CronEd.PR_TT*10))
rounded rectangle at (270,270)-(301,291): text "%.1f"; shows WORD_TO_REAL(CronEd.PR.Setpoint[30])/10; runs INTERN ASSIGN CronEd.PR.Setpoint[30]:=(REAL_TO_WORD(CronEd.PR_TT*10))
rounded rectangle at (270,290)-(301,311): text "%.1f"; shows WORD_TO_REAL(CronEd.PR.Setpoint[31])/10; runs INTERN ASSIGN CronEd.PR.Setpoint[31]:=(REAL_TO_WORD(CronEd.PR_TT*10))
rectangle at (270,200)-(301,221): text "h07"; runs INTERN ASSIGN CronEd.PR.Setpoint[31]:=(REAL_TO_WORD(CronEd.PR_TT*10));INTERN ASSIGN CronEd.PR.Setpoint[30]:=(REAL_TO_WORD(CronEd.PR_TT*10));INTERN ASSIGN CronEd.PR.Setpoint[29]:=(REAL_TO_WORD(CronEd.PR_TT*10));INTERN ASSIGN CronEd.PR.Setpoint[28]:=(REAL_TO_WORD(CronEd.PR_TT*10))
rounded rectangle at (300,230)-(331,251): text "%.1f"; shows WORD_TO_REAL(CronEd.PR.Setpoint[32])/10; runs INTERN ASSIGN CronEd.PR.Setpoint[32]:=(REAL_TO_WORD(CronEd.PR_TT*10))
rounded rectangle at (300,250)-(331,271): text "%.1f"; shows WORD_TO_REAL(CronEd.PR.Setpoint[33])/10; runs INTERN ASSIGN CronEd.PR.Setpoint[33]:=(REAL_TO_WORD(CronEd.PR_TT*10))
rounded rectangle at (300,270)-(331,291): text "%.1f"; shows WORD_TO_REAL(CronEd.PR.Setpoint[34])/10; runs INTERN ASSIGN CronEd.PR.Setpoint[34]:=(REAL_TO_WORD(CronEd.PR_TT*10))
rounded rectangle at (300,290)-(331,311): text "%.1f"; shows WORD_TO_REAL(CronEd.PR.Setpoint[35])/10; runs INTERN ASSIGN CronEd.PR.Setpoint[35]:=(REAL_TO_WORD(CronEd.PR_TT*10))
rectangle at (300,200)-(331,221): text "h08"; runs INTERN ASSIGN CronEd.PR.Setpoint[35]:=(REAL_TO_WORD(CronEd.PR_TT*10));INTERN ASSIGN CronEd.PR.Setpoint[34]:=(REAL_TO_WORD(CronEd.PR_TT*10));INTERN ASSIGN CronEd.PR.Setpoint[33]:=(REAL_TO_WORD(CronEd.PR_TT*10));INTERN ASSIGN CronEd.PR.Setpoint[32]:=(REAL_TO_WORD(CronEd.PR_TT*10))
rounded rectangle at (330,230)-(361,251): text "%.1f"; shows WORD_TO_REAL(CronEd.PR.Setpoint[36])/10; runs INTERN ASSIGN CronEd.PR.Setpoint[36]:=(REAL_TO_WORD(CronEd.PR_TT*10))
rounded rectangle at (330,250)-(361,271): text "%.1f"; shows WORD_TO_REAL(CronEd.PR.Setpoint[37])/10; runs INTERN ASSIGN CronEd.PR.Setpoint[37]:=(REAL_TO_WORD(CronEd.PR_TT*10))
rounded rectangle at (330,270)-(361,291): text "%.1f"; shows WORD_TO_REAL(CronEd.PR.Setpoint[38])/10; runs INTERN ASSIGN CronEd.PR.Setpoint[38]:=(REAL_TO_WORD(CronEd.PR_TT*10))
rounded rectangle at (330,290)-(361,311): text "%.1f"; shows WORD_TO_REAL(CronEd.PR.Setpoint[39])/10; runs INTERN ASSIGN CronEd.PR.Setpoint[39]:=(REAL_TO_WORD(CronEd.PR_TT*10))
rectangle at (330,200)-(361,221): text "h09"; runs INTERN ASSIGN CronEd.PR.Setpoint[39]:=(REAL_TO_WORD(CronEd.PR_TT*10));INTERN ASSIGN CronEd.PR.Setpoint[38]:=(REAL_TO_WORD(CronEd.PR_TT*10));INTERN ASSIGN CronEd.PR.Setpoint[37]:=(REAL_TO_WORD(CronEd.PR_TT*10));INTERN ASSIGN CronEd.PR.Setpoint[36]:=(REAL_TO_WORD(CronEd.PR_TT*10))
rounded rectangle at (360,230)-(391,251): text "%.1f"; shows WORD_TO_REAL(CronEd.PR.Setpoint[40])/10; runs INTERN ASSIGN CronEd.PR.Setpoint[40]:=(REAL_TO_WORD(CronEd.PR_TT*10))
rounded rectangle at (360,250)-(391,271): text "%.1f"; shows WORD_TO_REAL(CronEd.PR.Setpoint[41])/10; runs INTERN ASSIGN CronEd.PR.Setpoint[41]:=(REAL_TO_WORD(CronEd.PR_TT*10))
rounded rectangle at (360,270)-(391,291): text "%.1f"; shows WORD_TO_REAL(CronEd.PR.Setpoint[42])/10; runs INTERN ASSIGN CronEd.PR.Setpoint[42]:=(REAL_TO_WORD(CronEd.PR_TT*10))
rounded rectangle at (360,290)-(391,311): text "%.1f"; shows WORD_TO_REAL(CronEd.PR.Setpoint[43])/10; runs INTERN ASSIGN CronEd.PR.Setpoint[43]:=(REAL_TO_WORD(CronEd.PR_TT*10))
rectangle at (360,200)-(391,221): text "h10"; runs INTERN ASSIGN CronEd.PR.Setpoint[43]:=(REAL_TO_WORD(CronEd.PR_TT*10));INTERN ASSIGN CronEd.PR.Setpoint[42]:=(REAL_TO_WORD(CronEd.PR_TT*10));INTERN ASSIGN CronEd.PR.Setpoint[41]:=(REAL_TO_WORD(CronEd.PR_TT*10));INTERN ASSIGN CronEd.PR.Setpoint[40]:=(REAL_TO_WORD(CronEd.PR_TT*10))
rounded rectangle at (390,230)-(421,251): text "%.1f"; shows WORD_TO_REAL(CronEd.PR.Setpoint[44])/10; runs INTERN ASSIGN CronEd.PR.Setpoint[44]:=(REAL_TO_WORD(CronEd.PR_TT*10))
rounded rectangle at (390,250)-(421,271): text "%.1f"; shows WORD_TO_REAL(CronEd.PR.Setpoint[45])/10; runs INTERN ASSIGN CronEd.PR.Setpoint[45]:=(REAL_TO_WORD(CronEd.PR_TT*10))
rounded rectangle at (390,270)-(421,291): text "%.1f"; shows WORD_TO_REAL(CronEd.PR.Setpoint[46])/10; runs INTERN ASSIGN CronEd.PR.Setpoint[46]:=(REAL_TO_WORD(CronEd.PR_TT*10))
rounded rectangle at (390,290)-(421,311): text "%.1f"; shows WORD_TO_REAL(CronEd.PR.Setpoint[47])/10; runs INTERN ASSIGN CronEd.PR.Setpoint[47]:=(REAL_TO_WORD(CronEd.PR_TT*10))
rectangle at (390,200)-(421,221): text "h11"; runs INTERN ASSIGN CronEd.PR.Setpoint[47]:=(REAL_TO_WORD(CronEd.PR_TT*10));INTERN ASSIGN CronEd.PR.Setpoint[46]:=(REAL_TO_WORD(CronEd.PR_TT*10));INTERN ASSIGN CronEd.PR.Setpoint[45]:=(REAL_TO_WORD(CronEd.PR_TT*10));INTERN ASSIGN CronEd.PR.Setpoint[44]:=(REAL_TO_WORD(CronEd.PR_TT*10))
rounded rectangle at (420,230)-(451,251): text "%.1f"; shows WORD_TO_REAL(CronEd.PR.Setpoint[48])/10; runs INTERN ASSIGN CronEd.PR.Setpoint[48]:=(REAL_TO_WORD(CronEd.PR_TT*10))
rounded rectangle at (420,250)-(451,271): text "%.1f"; shows WORD_TO_REAL(CronEd.PR.Setpoint[49])/10; runs INTERN ASSIGN CronEd.PR.Setpoint[49]:=(REAL_TO_WORD(CronEd.PR_TT*10))
rounded rectangle at (420,270)-(451,291): text "%.1f"; shows WORD_TO_REAL(CronEd.PR.Setpoint[50])/10; runs INTERN ASSIGN CronEd.PR.Setpoint[50]:=(REAL_TO_WORD(CronEd.PR_TT*10))
rounded rectangle at (420,290)-(451,311): text "%.1f"; shows WORD_TO_REAL(CronEd.PR.Setpoint[51])/10; runs INTERN ASSIGN CronEd.PR.Setpoint[51]:=(REAL_TO_WORD(CronEd.PR_TT*10))
rectangle at (420,200)-(451,221): text "h12"; runs INTERN ASSIGN CronEd.PR.Setpoint[51]:=(REAL_TO_WORD(CronEd.PR_TT*10));INTERN ASSIGN CronEd.PR.Setpoint[50]:=(REAL_TO_WORD(CronEd.PR_TT*10));INTERN ASSIGN CronEd.PR.Setpoint[49]:=(REAL_TO_WORD(CronEd.PR_TT*10));INTERN ASSIGN CronEd.PR.Setpoint[48]:=(REAL_TO_WORD(CronEd.PR_TT*10))
rounded rectangle at (450,230)-(481,251): text "%.1f"; shows WORD_TO_REAL(CronEd.PR.Setpoint[52])/10; runs INTERN ASSIGN CronEd.PR.Setpoint[52]:=(REAL_TO_WORD(CronEd.PR_TT*10))
rounded rectangle at (450,250)-(481,271): text "%.1f"; shows WORD_TO_REAL(CronEd.PR.Setpoint[53])/10; runs INTERN ASSIGN CronEd.PR.Setpoint[53]:=(REAL_TO_WORD(CronEd.PR_TT*10))
rounded rectangle at (450,270)-(481,291): text "%.1f"; shows WORD_TO_REAL(CronEd.PR.Setpoint[54])/10; runs INTERN ASSIGN CronEd.PR.Setpoint[54]:=(REAL_TO_WORD(CronEd.PR_TT*10))
rounded rectangle at (450,290)-(481,311): text "%.1f"; shows WORD_TO_REAL(CronEd.PR.Setpoint[55])/10; runs INTERN ASSIGN CronEd.PR.Setpoint[55]:=(REAL_TO_WORD(CronEd.PR_TT*10))
rectangle at (450,200)-(481,221): text "h13"; runs INTERN ASSIGN CronEd.PR.Setpoint[55]:=(REAL_TO_WORD(CronEd.PR_TT*10));INTERN ASSIGN CronEd.PR.Setpoint[54]:=(REAL_TO_WORD(CronEd.PR_TT*10));INTERN ASSIGN CronEd.PR.Setpoint[53]:=(REAL_TO_WORD(CronEd.PR_TT*10));INTERN ASSIGN CronEd.PR.Setpoint[52]:=(REAL_TO_WORD(CronEd.PR_TT*10))
rounded rectangle at (480,230)-(511,251): text "%.1f"; shows WORD_TO_REAL(CronEd.PR.Setpoint[56])/10; runs INTERN ASSIGN CronEd.PR.Setpoint[56]:=(REAL_TO_WORD(CronEd.PR_TT*10))
rounded rectangle at (480,250)-(511,271): text "%.1f"; shows WORD_TO_REAL(CronEd.PR.Setpoint[57])/10; runs INTERN ASSIGN CronEd.PR.Setpoint[57]:=(REAL_TO_WORD(CronEd.PR_TT*10))
rounded rectangle at (480,270)-(511,291): text "%.1f"; shows WORD_TO_REAL(CronEd.PR.Setpoint[58])/10; runs INTERN ASSIGN CronEd.PR.Setpoint[58]:=(REAL_TO_WORD(CronEd.PR_TT*10))
rounded rectangle at (480,290)-(511,311): text "%.1f"; shows WORD_TO_REAL(CronEd.PR.Setpoint[59])/10; runs INTERN ASSIGN CronEd.PR.Setpoint[59]:=(REAL_TO_WORD(CronEd.PR_TT*10))
rectangle at (480,200)-(511,221): text "h14"; runs INTERN ASSIGN CronEd.PR.Setpoint[59]:=(REAL_TO_WORD(CronEd.PR_TT*10));INTERN ASSIGN CronEd.PR.Setpoint[58]:=(REAL_TO_WORD(CronEd.PR_TT*10));INTERN ASSIGN CronEd.PR.Setpoint[57]:=(REAL_TO_WORD(CronEd.PR_TT*10));INTERN ASSIGN CronEd.PR.Setpoint[56]:=(REAL_TO_WORD(CronEd.PR_TT*10))
rounded rectangle at (510,230)-(541,251): text "%.1f"; shows WORD_TO_REAL(CronEd.PR.Setpoint[60])/10; runs INTERN ASSIGN CronEd.PR.Setpoint[60]:=(REAL_TO_WORD(CronEd.PR_TT*10))
rounded rectangle at (510,250)-(541,271): text "%.1f"; shows WORD_TO_REAL(CronEd.PR.Setpoint[61])/10; runs INTERN ASSIGN CronEd.PR.Setpoint[61]:=(REAL_TO_WORD(CronEd.PR_TT*10))
rounded rectangle at (510,270)-(541,291): text "%.1f"; shows WORD_TO_REAL(CronEd.PR.Setpoint[62])/10; runs INTERN ASSIGN CronEd.PR.Setpoint[62]:=(REAL_TO_WORD(CronEd.PR_TT*10))
rounded rectangle at (510,290)-(541,311): text "%.1f"; shows WORD_TO_REAL(CronEd.PR.Setpoint[63])/10; runs INTERN ASSIGN CronEd.PR.Setpoint[63]:=(REAL_TO_WORD(CronEd.PR_TT*10))
rectangle at (510,200)-(541,221): text "h15"; runs INTERN ASSIGN CronEd.PR.Setpoint[63]:=(REAL_TO_WORD(CronEd.PR_TT*10));INTERN ASSIGN CronEd.PR.Setpoint[62]:=(REAL_TO_WORD(CronEd.PR_TT*10));INTERN ASSIGN CronEd.PR.Setpoint[61]:=(REAL_TO_WORD(CronEd.PR_TT*10));INTERN ASSIGN CronEd.PR.Setpoint[60]:=(REAL_TO_WORD(CronEd.PR_TT*10))
rounded rectangle at (540,230)-(571,251): text "%.1f"; shows WORD_TO_REAL(CronEd.PR.Setpoint[64])/10; runs INTERN ASSIGN CronEd.PR.Setpoint[64]:=(REAL_TO_WORD(CronEd.PR_TT*10))
rounded rectangle at (540,250)-(571,271): text "%.1f"; shows WORD_TO_REAL(CronEd.PR.Setpoint[65])/10; runs INTERN ASSIGN CronEd.PR.Setpoint[65]:=(REAL_TO_WORD(CronEd.PR_TT*10))
rounded rectangle at (540,270)-(571,291): text "%.1f"; shows WORD_TO_REAL(CronEd.PR.Setpoint[66])/10; runs INTERN ASSIGN CronEd.PR.Setpoint[66]:=(REAL_TO_WORD(CronEd.PR_TT*10))
rounded rectangle at (540,290)-(571,311): text "%.1f"; shows WORD_TO_REAL(CronEd.PR.Setpoint[67])/10; runs INTERN ASSIGN CronEd.PR.Setpoint[67]:=(REAL_TO_WORD(CronEd.PR_TT*10))
rectangle at (540,200)-(571,221): text "h16"; runs INTERN ASSIGN CronEd.PR.Setpoint[67]:=(REAL_TO_WORD(CronEd.PR_TT*10));INTERN ASSIGN CronEd.PR.Setpoint[66]:=(REAL_TO_WORD(CronEd.PR_TT*10));INTERN ASSIGN CronEd.PR.Setpoint[65]:=(REAL_TO_WORD(CronEd.PR_TT*10));INTERN ASSIGN CronEd.PR.Setpoint[64]:=(REAL_TO_WORD(CronEd.PR_TT*10))
rounded rectangle at (570,230)-(601,251): text "%.1f"; shows WORD_TO_REAL(CronEd.PR.Setpoint[68])/10; runs INTERN ASSIGN CronEd.PR.Setpoint[68]:=(REAL_TO_WORD(CronEd.PR_TT*10))
rounded rectangle at (570,250)-(601,271): text "%.1f"; shows WORD_TO_REAL(CronEd.PR.Setpoint[69])/10; runs INTERN ASSIGN CronEd.PR.Setpoint[69]:=(REAL_TO_WORD(CronEd.PR_TT*10))
rounded rectangle at (570,270)-(601,291): text "%.1f"; shows WORD_TO_REAL(CronEd.PR.Setpoint[70])/10; runs INTERN ASSIGN CronEd.PR.Setpoint[70]:=(REAL_TO_WORD(CronEd.PR_TT*10))
rounded rectangle at (570,290)-(601,311): text "%.1f"; shows WORD_TO_REAL(CronEd.PR.Setpoint[71])/10; runs INTERN ASSIGN CronEd.PR.Setpoint[71]:=(REAL_TO_WORD(CronEd.PR_TT*10))
rectangle at (570,200)-(601,221): text "h17"; runs INTERN ASSIGN CronEd.PR.Setpoint[71]:=(REAL_TO_WORD(CronEd.PR_TT*10));INTERN ASSIGN CronEd.PR.Setpoint[70]:=(REAL_TO_WORD(CronEd.PR_TT*10));INTERN ASSIGN CronEd.PR.Setpoint[69]:=(REAL_TO_WORD(CronEd.PR_TT*10));INTERN ASSIGN CronEd.PR.Setpoint[68]:=(REAL_TO_WORD(CronEd.PR_TT*10))
rounded rectangle at (600,230)-(631,251): text "%.1f"; shows WORD_TO_REAL(CronEd.PR.Setpoint[72])/10; runs INTERN ASSIGN CronEd.PR.Setpoint[72]:=(REAL_TO_WORD(CronEd.PR_TT*10))
rounded rectangle at (600,250)-(631,271): text "%.1f"; shows WORD_TO_REAL(CronEd.PR.Setpoint[73])/10; runs INTERN ASSIGN CronEd.PR.Setpoint[73]:=(REAL_TO_WORD(CronEd.PR_TT*10))
rounded rectangle at (600,270)-(631,291): text "%.1f"; shows WORD_TO_REAL(CronEd.PR.Setpoint[74])/10; runs INTERN ASSIGN CronEd.PR.Setpoint[74]:=(REAL_TO_WORD(CronEd.PR_TT*10))
rounded rectangle at (600,290)-(631,311): text "%.1f"; shows WORD_TO_REAL(CronEd.PR.Setpoint[75])/10; runs INTERN ASSIGN CronEd.PR.Setpoint[75]:=(REAL_TO_WORD(CronEd.PR_TT*10))
rectangle at (600,200)-(631,221): text "h18"; runs INTERN ASSIGN CronEd.PR.Setpoint[75]:=(REAL_TO_WORD(CronEd.PR_TT*10));INTERN ASSIGN CronEd.PR.Setpoint[74]:=(REAL_TO_WORD(CronEd.PR_TT*10));INTERN ASSIGN CronEd.PR.Setpoint[73]:=(REAL_TO_WORD(CronEd.PR_TT*10));INTERN ASSIGN CronEd.PR.Setpoint[72]:=(REAL_TO_WORD(CronEd.PR_TT*10))
rounded rectangle at (630,230)-(661,251): text "%.1f"; shows WORD_TO_REAL(CronEd.PR.Setpoint[76])/10; runs INTERN ASSIGN CronEd.PR.Setpoint[76]:=(REAL_TO_WORD(CronEd.PR_TT*10))
rounded rectangle at (630,250)-(661,271): text "%.1f"; shows WORD_TO_REAL(CronEd.PR.Setpoint[77])/10; runs INTERN ASSIGN CronEd.PR.Setpoint[77]:=(REAL_TO_WORD(CronEd.PR_TT*10))
rounded rectangle at (630,270)-(661,291): text "%.1f"; shows WORD_TO_REAL(CronEd.PR.Setpoint[78])/10; runs INTERN ASSIGN CronEd.PR.Setpoint[78]:=(REAL_TO_WORD(CronEd.PR_TT*10))
rounded rectangle at (630,290)-(661,311): text "%.1f"; shows WORD_TO_REAL(CronEd.PR.Setpoint[79])/10; runs INTERN ASSIGN CronEd.PR.Setpoint[79]:=(REAL_TO_WORD(CronEd.PR_TT*10))
rectangle at (630,200)-(661,221): text "h19"; runs INTERN ASSIGN CronEd.PR.Setpoint[79]:=(REAL_TO_WORD(CronEd.PR_TT*10));INTERN ASSIGN CronEd.PR.Setpoint[78]:=(REAL_TO_WORD(CronEd.PR_TT*10));INTERN ASSIGN CronEd.PR.Setpoint[77]:=(REAL_TO_WORD(CronEd.PR_TT*10));INTERN ASSIGN CronEd.PR.Setpoint[76]:=(REAL_TO_WORD(CronEd.PR_TT*10))
rounded rectangle at (660,230)-(691,251): text "%.1f"; shows WORD_TO_REAL(CronEd.PR.Setpoint[80])/10; runs INTERN ASSIGN CronEd.PR.Setpoint[80]:=(REAL_TO_WORD(CronEd.PR_TT*10))
rounded rectangle at (660,250)-(691,271): text "%.1f"; shows WORD_TO_REAL(CronEd.PR.Setpoint[81])/10; runs INTERN ASSIGN CronEd.PR.Setpoint[81]:=(REAL_TO_WORD(CronEd.PR_TT*10))
rounded rectangle at (660,270)-(691,291): text "%.1f"; shows WORD_TO_REAL(CronEd.PR.Setpoint[82])/10; runs INTERN ASSIGN CronEd.PR.Setpoint[82]:=(REAL_TO_WORD(CronEd.PR_TT*10))
rounded rectangle at (660,290)-(691,311): text "%.1f"; shows WORD_TO_REAL(CronEd.PR.Setpoint[83])/10; runs INTERN ASSIGN CronEd.PR.Setpoint[83]:=(REAL_TO_WORD(CronEd.PR_TT*10))
rectangle at (660,200)-(691,221): text "h20"; runs INTERN ASSIGN CronEd.PR.Setpoint[83]:=(REAL_TO_WORD(CronEd.PR_TT*10));INTERN ASSIGN CronEd.PR.Setpoint[82]:=(REAL_TO_WORD(CronEd.PR_TT*10));INTERN ASSIGN CronEd.PR.Setpoint[81]:=(REAL_TO_WORD(CronEd.PR_TT*10));INTERN ASSIGN CronEd.PR.Setpoint[80]:=(REAL_TO_WORD(CronEd.PR_TT*10))
rounded rectangle at (690,230)-(721,251): text "%.1f"; shows WORD_TO_REAL(CronEd.PR.Setpoint[84])/10; runs INTERN ASSIGN CronEd.PR.Setpoint[84]:=(REAL_TO_WORD(CronEd.PR_TT*10))
rounded rectangle at (690,250)-(721,271): text "%.1f"; shows WORD_TO_REAL(CronEd.PR.Setpoint[85])/10; runs INTERN ASSIGN CronEd.PR.Setpoint[85]:=(REAL_TO_WORD(CronEd.PR_TT*10))
rounded rectangle at (690,270)-(721,291): text "%.1f"; shows WORD_TO_REAL(CronEd.PR.Setpoint[86])/10; runs INTERN ASSIGN CronEd.PR.Setpoint[86]:=(REAL_TO_WORD(CronEd.PR_TT*10))
rounded rectangle at (690,290)-(721,311): text "%.1f"; shows WORD_TO_REAL(CronEd.PR.Setpoint[87])/10; runs INTERN ASSIGN CronEd.PR.Setpoint[87]:=(REAL_TO_WORD(CronEd.PR_TT*10))
rectangle at (690,200)-(721,221): text "h21"; runs INTERN ASSIGN CronEd.PR.Setpoint[87]:=(REAL_TO_WORD(CronEd.PR_TT*10));INTERN ASSIGN CronEd.PR.Setpoint[86]:=(REAL_TO_WORD(CronEd.PR_TT*10));INTERN ASSIGN CronEd.PR.Setpoint[85]:=(REAL_TO_WORD(CronEd.PR_TT*10));INTERN ASSIGN CronEd.PR.Setpoint[84]:=(REAL_TO_WORD(CronEd.PR_TT*10))
rounded rectangle at (720,230)-(751,251): text "%.1f"; shows WORD_TO_REAL(CronEd.PR.Setpoint[88])/10; runs INTERN ASSIGN CronEd.PR.Setpoint[88]:=(REAL_TO_WORD(CronEd.PR_TT*10))
rounded rectangle at (720,250)-(751,271): text "%.1f"; shows WORD_TO_REAL(CronEd.PR.Setpoint[89])/10; runs INTERN ASSIGN CronEd.PR.Setpoint[89]:=(REAL_TO_WORD(CronEd.PR_TT*10))
rounded rectangle at (720,270)-(751,291): text "%.1f"; shows WORD_TO_REAL(CronEd.PR.Setpoint[90])/10; runs INTERN ASSIGN CronEd.PR.Setpoint[90]:=(REAL_TO_WORD(CronEd.PR_TT*10))
rounded rectangle at (720,290)-(751,311): text "%.1f"; shows WORD_TO_REAL(CronEd.PR.Setpoint[91])/10; runs INTERN ASSIGN CronEd.PR.Setpoint[91]:=(REAL_TO_WORD(CronEd.PR_TT*10))
rectangle at (720,200)-(751,221): text "h22"; runs INTERN ASSIGN CronEd.PR.Setpoint[91]:=(REAL_TO_WORD(CronEd.PR_TT*10));INTERN ASSIGN CronEd.PR.Setpoint[90]:=(REAL_TO_WORD(CronEd.PR_TT*10));INTERN ASSIGN CronEd.PR.Setpoint[89]:=(REAL_TO_WORD(CronEd.PR_TT*10));INTERN ASSIGN CronEd.PR.Setpoint[88]:=(REAL_TO_WORD(CronEd.PR_TT*10))
rounded rectangle at (750,230)-(781,251): text "%.1f"; shows WORD_TO_REAL(CronEd.PR.Setpoint[92])/10; runs INTERN ASSIGN CronEd.PR.Setpoint[92]:=(REAL_TO_WORD(CronEd.PR_TT*10))
rounded rectangle at (750,250)-(781,271): text "%.1f"; shows WORD_TO_REAL(CronEd.PR.Setpoint[93])/10; runs INTERN ASSIGN CronEd.PR.Setpoint[93]:=(REAL_TO_WORD(CronEd.PR_TT*10))
rounded rectangle at (750,270)-(781,291): text "%.1f"; shows WORD_TO_REAL(CronEd.PR.Setpoint[94])/10; runs INTERN ASSIGN CronEd.PR.Setpoint[94]:=(REAL_TO_WORD(CronEd.PR_TT*10))
rounded rectangle at (750,290)-(781,311): text "%.1f"; shows WORD_TO_REAL(CronEd.PR.Setpoint[95])/10; runs INTERN ASSIGN CronEd.PR.Setpoint[95]:=(REAL_TO_WORD(CronEd.PR_TT*10))
rectangle at (750,200)-(781,221): text "h23"; runs INTERN ASSIGN CronEd.PR.Setpoint[95]:=(REAL_TO_WORD(CronEd.PR_TT*10));INTERN ASSIGN CronEd.PR.Setpoint[94]:=(REAL_TO_WORD(CronEd.PR_TT*10));INTERN ASSIGN CronEd.PR.Setpoint[93]:=(REAL_TO_WORD(CronEd.PR_TT*10));INTERN ASSIGN CronEd.PR.Setpoint[92]:=(REAL_TO_WORD(CronEd.PR_TT*10))
rectangle at (410,360)-(491,381): text "Month"
rectangle at (490,360)-(531,381): text "%d"; shows CronEd.CA_Sel; alarm colour if CronEd.CA_Sel<>CronEd.CA_Act; editable 1..12
rectangle at (410,390)-(491,411): text "Profile Nr."
rectangle at (490,390)-(531,411): text "%d"; shows CronEd.CA_TPR; editable 0..10
button at (540,360)-(601,381): text "Load"; toggles CronEd.CA_Load
button at (610,360)-(671,381): text "Save"; toggles CronEd.CA_Save
rounded rectangle at (160,360)-(191,381): text "%d"; shows CronEd.CA.Profile[0]; invisible if CronEd.CA_DayF>0; alarm colour if CronEd.CA.Profile[0]=0; runs INTERN ASSIGN CronEd.CA.Profile[0]:=(CronEd.CA_TPR)
rectangle at (120,360)-(151,381): text "1"
rounded rectangle at (190,360)-(221,381): text "%d"; shows CronEd.CA.Profile[1]; invisible if CronEd.CA_DayF>1; alarm colour if CronEd.CA.Profile[1]=0; runs INTERN ASSIGN CronEd.CA.Profile[1]:=(CronEd.CA_TPR)
rounded rectangle at (220,360)-(251,381): text "%d"; shows CronEd.CA.Profile[2]; invisible if CronEd.CA_DayF>2; alarm colour if CronEd.CA.Profile[2]=0; runs INTERN ASSIGN CronEd.CA.Profile[2]:=(CronEd.CA_TPR)
rounded rectangle at (250,360)-(281,381): text "%d"; shows CronEd.CA.Profile[3]; invisible if CronEd.CA_DayF>3; alarm colour if CronEd.CA.Profile[3]=0; runs INTERN ASSIGN CronEd.CA.Profile[3]:=(CronEd.CA_TPR)
rounded rectangle at (280,360)-(311,381): text "%d"; shows CronEd.CA.Profile[4]; invisible if CronEd.CA_DayF>4; alarm colour if CronEd.CA.Profile[4]=0; runs INTERN ASSIGN CronEd.CA.Profile[4]:=(CronEd.CA_TPR)
rounded rectangle at (310,360)-(341,381): text "%d"; shows CronEd.CA.Profile[5]; invisible if CronEd.CA_DayF>5; alarm colour if CronEd.CA.Profile[5]=0; runs INTERN ASSIGN CronEd.CA.Profile[5]:=(CronEd.CA_TPR)
rounded rectangle at (340,360)-(371,381): text "%d"; shows CronEd.CA.Profile[6]; alarm colour if CronEd.CA.Profile[6]=0; runs INTERN ASSIGN CronEd.CA.Profile[6]:=(CronEd.CA_TPR)
rounded rectangle at (160,380)-(191,401): text "%d"; shows CronEd.CA.Profile[7]; alarm colour if CronEd.CA.Profile[7]=0; runs INTERN ASSIGN CronEd.CA.Profile[7]:=(CronEd.CA_TPR)
rectangle at (120,380)-(151,401): text "8"
rounded rectangle at (190,380)-(221,401): text "%d"; shows CronEd.CA.Profile[8]; alarm colour if CronEd.CA.Profile[8]=0; runs INTERN ASSIGN CronEd.CA.Profile[8]:=(CronEd.CA_TPR)
rounded rectangle at (220,380)-(251,401): text "%d"; shows CronEd.CA.Profile[9]; alarm colour if CronEd.CA.Profile[9]=0; runs INTERN ASSIGN CronEd.CA.Profile[9]:=(CronEd.CA_TPR)
rounded rectangle at (250,380)-(281,401): text "%d"; shows CronEd.CA.Profile[10]; alarm colour if CronEd.CA.Profile[10]=0; runs INTERN ASSIGN CronEd.CA.Profile[10]:=(CronEd.CA_TPR)
rounded rectangle at (280,380)-(311,401): text "%d"; shows CronEd.CA.Profile[11]; alarm colour if CronEd.CA.Profile[11]=0; runs INTERN ASSIGN CronEd.CA.Profile[11]:=(CronEd.CA_TPR)
rounded rectangle at (310,380)-(341,401): text "%d"; shows CronEd.CA.Profile[12]; alarm colour if CronEd.CA.Profile[12]=0; runs INTERN ASSIGN CronEd.CA.Profile[12]:=(CronEd.CA_TPR)
rounded rectangle at (340,380)-(371,401): text "%d"; shows CronEd.CA.Profile[13]; alarm colour if CronEd.CA.Profile[13]=0; runs INTERN ASSIGN CronEd.CA.Profile[13]:=(CronEd.CA_TPR)
rounded rectangle at (160,400)-(191,421): text "%d"; shows CronEd.CA.Profile[14]; alarm colour if CronEd.CA.Profile[14]=0; runs INTERN ASSIGN CronEd.CA.Profile[14]:=(CronEd.CA_TPR)
rectangle at (120,400)-(151,421): text "15"
rounded rectangle at (190,400)-(221,421): text "%d"; shows CronEd.CA.Profile[15]; alarm colour if CronEd.CA.Profile[15]=0; runs INTERN ASSIGN CronEd.CA.Profile[15]:=(CronEd.CA_TPR)
rounded rectangle at (220,400)-(251,421): text "%d"; shows CronEd.CA.Profile[16]; alarm colour if CronEd.CA.Profile[16]=0; runs INTERN ASSIGN CronEd.CA.Profile[16]:=(CronEd.CA_TPR)
rounded rectangle at (250,400)-(281,421): text "%d"; shows CronEd.CA.Profile[17]; alarm colour if CronEd.CA.Profile[17]=0; runs INTERN ASSIGN CronEd.CA.Profile[17]:=(CronEd.CA_TPR)
rounded rectangle at (280,400)-(311,421): text "%d"; shows CronEd.CA.Profile[18]; alarm colour if CronEd.CA.Profile[18]=0; runs INTERN ASSIGN CronEd.CA.Profile[18]:=(CronEd.CA_TPR)
rounded rectangle at (310,400)-(341,421): text "%d"; shows CronEd.CA.Profile[19]; alarm colour if CronEd.CA.Profile[19]=0; runs INTERN ASSIGN CronEd.CA.Profile[19]:=(CronEd.CA_TPR)
rounded rectangle at (340,400)-(371,421): text "%d"; shows CronEd.CA.Profile[20]; alarm colour if CronEd.CA.Profile[20]=0; runs INTERN ASSIGN CronEd.CA.Profile[20]:=(CronEd.CA_TPR)
rounded rectangle at (160,420)-(191,441): text "%d"; shows CronEd.CA.Profile[21]; alarm colour if CronEd.CA.Profile[21]=0; runs INTERN ASSIGN CronEd.CA.Profile[21]:=(CronEd.CA_TPR)
rectangle at (120,420)-(151,441): text "22"
rounded rectangle at (190,420)-(221,441): text "%d"; shows CronEd.CA.Profile[22]; alarm colour if CronEd.CA.Profile[22]=0; runs INTERN ASSIGN CronEd.CA.Profile[22]:=(CronEd.CA_TPR)
rounded rectangle at (220,420)-(251,441): text "%d"; shows CronEd.CA.Profile[23]; alarm colour if CronEd.CA.Profile[23]=0; runs INTERN ASSIGN CronEd.CA.Profile[23]:=(CronEd.CA_TPR)
rounded rectangle at (250,420)-(281,441): text "%d"; shows CronEd.CA.Profile[24]; alarm colour if CronEd.CA.Profile[24]=0; runs INTERN ASSIGN CronEd.CA.Profile[24]:=(CronEd.CA_TPR)
rounded rectangle at (280,420)-(311,441): text "%d"; shows CronEd.CA.Profile[25]; alarm colour if CronEd.CA.Profile[25]=0; runs INTERN ASSIGN CronEd.CA.Profile[25]:=(CronEd.CA_TPR)
rounded rectangle at (310,420)-(341,441): text "%d"; shows CronEd.CA.Profile[26]; alarm colour if CronEd.CA.Profile[26]=0; runs INTERN ASSIGN CronEd.CA.Profile[26]:=(CronEd.CA_TPR)
rounded rectangle at (340,420)-(371,441): text "%d"; shows CronEd.CA.Profile[27]; alarm colour if CronEd.CA.Profile[27]=0; runs INTERN ASSIGN CronEd.CA.Profile[27]:=(CronEd.CA_TPR)
rounded rectangle at (160,440)-(191,461): text "%d"; shows CronEd.CA.Profile[28]; alarm colour if CronEd.CA.Profile[28]=0; runs INTERN ASSIGN CronEd.CA.Profile[28]:=(CronEd.CA_TPR)
rectangle at (120,440)-(151,461): text "29"
rounded rectangle at (190,440)-(221,461): text "%d"; shows CronEd.CA.Profile[29]; alarm colour if CronEd.CA.Profile[29]=0; runs INTERN ASSIGN CronEd.CA.Profile[29]:=(CronEd.CA_TPR)
rounded rectangle at (220,440)-(251,461): text "%d"; shows CronEd.CA.Profile[30]; alarm colour if CronEd.CA.Profile[30]=0; runs INTERN ASSIGN CronEd.CA.Profile[30]:=(CronEd.CA_TPR)
rounded rectangle at (250,440)-(281,461): text "%d"; shows CronEd.CA.Profile[31]; alarm colour if CronEd.CA.Profile[31]=0; runs INTERN ASSIGN CronEd.CA.Profile[31]:=(CronEd.CA_TPR)
rounded rectangle at (280,440)-(311,461): text "%d"; shows CronEd.CA.Profile[32]; invisible if CronEd.CA_DayL<32; alarm colour if CronEd.CA.Profile[32]=0; runs INTERN ASSIGN CronEd.CA.Profile[32]:=(CronEd.CA_TPR)
rounded rectangle at (310,440)-(341,461): text "%d"; shows CronEd.CA.Profile[33]; invisible if CronEd.CA_DayL<33; alarm colour if CronEd.CA.Profile[33]=0; runs INTERN ASSIGN CronEd.CA.Profile[33]:=(CronEd.CA_TPR)
rounded rectangle at (340,440)-(371,461): text "%d"; shows CronEd.CA.Profile[34]; invisible if CronEd.CA_DayL<34; alarm colour if CronEd.CA.Profile[34]=0; runs INTERN ASSIGN CronEd.CA.Profile[34]:=(CronEd.CA_TPR)
rounded rectangle at (160,460)-(191,481): text "%d"; shows CronEd.CA.Profile[35]; invisible if CronEd.CA_DayL<35; alarm colour if CronEd.CA.Profile[35]=0; runs INTERN ASSIGN CronEd.CA.Profile[35]:=(CronEd.CA_TPR)
rectangle at (120,460)-(151,481): text "36"; invisible if CronEd.CA_DayL<35
rounded rectangle at (190,460)-(221,481): text "%d"; shows CronEd.CA.Profile[36]; invisible if CronEd.CA_DayL<36; alarm colour if CronEd.CA.Profile[36]=0; runs INTERN ASSIGN CronEd.CA.Profile[36]:=(CronEd.CA_TPR)
rounded rectangle at (220,460)-(251,481): text "%d"; shows CronEd.CA.Profile[37]; invisible if CronEd.CA_DayL<37; alarm colour if CronEd.CA.Profile[37]=0; runs INTERN ASSIGN CronEd.CA.Profile[37]:=(CronEd.CA_TPR)
rounded rectangle at (250,460)-(281,481): text "%d"; shows CronEd.CA.Profile[38]; invisible if CronEd.CA_DayL<38; alarm colour if CronEd.CA.Profile[38]=0; runs INTERN ASSIGN CronEd.CA.Profile[38]:=(CronEd.CA_TPR)
rounded rectangle at (280,460)-(311,481): text "%d"; shows CronEd.CA.Profile[39]; invisible if CronEd.CA_DayL<39; alarm colour if CronEd.CA.Profile[39]=0; runs INTERN ASSIGN CronEd.CA.Profile[39]:=(CronEd.CA_TPR)
rounded rectangle at (310,460)-(341,481): text "%d"; shows CronEd.CA.Profile[40]; invisible if CronEd.CA_DayL<40; alarm colour if CronEd.CA.Profile[40]=0; runs INTERN ASSIGN CronEd.CA.Profile[40]:=(CronEd.CA_TPR)
rounded rectangle at (340,460)-(371,481): text "%d"; shows CronEd.CA.Profile[41]; invisible if CronEd.CA_DayL<41; alarm colour if CronEd.CA.Profile[41]=0; runs INTERN ASSIGN CronEd.CA.Profile[41]:=(CronEd.CA_TPR)
rectangle at (310,60)-(371,81): text "Year"
rectangle at (370,60)-(411,81): text "%d"; shows CronEd.CN_YSel; alarm colour if CronEd.CN_YSel<>CronEd.CN_YAct; editable 2000..2100
rectangle at (480,60)-(761,81): text "%s"; shows CronEd.Message
button at (10,50)-(71,81): text "REINIT"; runs INTERN ASSIGN THER01.InitOK:=(FALSE);INTERN ASSIGN THER02.InitOK:=(FALSE);INTERN ASSIGN THER03.InitOK:=(FALSE);INTERN ASSIGN THER04.InitOK:=(FALSE);INTERN ASSIGN THER05.InitOK:=(FALSE)
2 more shapes without text or variables
*)

(* Visualisation VIS_SET
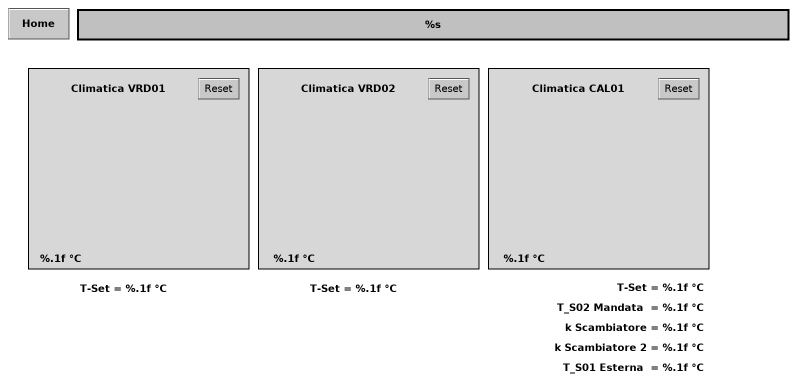
rectangle at (40,80)-(201,101): text "Climatica VRD01"
button at (200,80)-(241,101): text "Reset"; taps .VRD01.CLIM.InitOK
button at (10,10)-(71,41): text "Home"; opens PLC_VISU
rectangle at (80,280)-(221,301): text "T-Set = %.1f °C"; shows INT_TO_REAL(.VRD01.Ctrl_SetPoint)/10
rectangle at (270,80)-(431,101): text "Climatica VRD02"
button at (430,80)-(471,101): text "Reset"; taps .VRD02.CLIM.InitOK; runs INTERN ASSIGN VRD02_Clima.InitOK:=(FALSE)
rectangle at (310,280)-(451,301): text "T-Set = %.1f °C"; shows INT_TO_REAL(.VRD02.Ctrl_SetPoint)/10
rectangle at (40,250)-(91,271): text "%.1f °C"; shows INT_TO_REAL(.TPV05.IN)/10
rectangle at (270,250)-(321,271): text "%.1f °C"; shows INT_TO_REAL(.TPV06.IN)/10
rectangle at (500,80)-(661,101): text "Climatica CAL01"
button at (660,80)-(701,101): text "Reset"; taps .CAL01.CLIM.InitOK; runs INTERN ASSIGN VRD02_Clima.InitOK:=(FALSE)
rectangle at (500,250)-(551,271): text "%.1f °C"; shows INT_TO_REAL(.TPV06.IN)/10
rectangle at (79,11)-(791,42): text "%s"; shows .Plant_NAME
rectangle at (567,279)-(708,300): text "T-Set = %.1f °C"; shows INT_TO_REAL(.CAL01.SetPoint)/10
rectangle at (547,319)-(708,340): text "k Scambiatore = %.1f °C"; shows INT_TO_REAL(.OffsetSetPointManuale/10)
rectangle at (547,339)-(708,360): text "k Scambiatore 2 = %.1f °C"; shows INT_TO_REAL(.OffsetSetPointManuale2/10)
rectangle at (537,359)-(708,380): text "T_S01 Esterna  = %.1f °C"; shows INT_TO_REAL(.TPV01.IN)/10
rectangle at (547,299)-(708,320): text "T_S02 Mandata  = %.1f °C"; shows INT_TO_REAL(.TPV02.AVG)/10
3 more shapes without text or variables
44 elements of other kinds (tables, trends, ...) not read
*)
